// --- Comprobar que hay algo para generar
      L     "DB830_Dispositivos".Dispositivos[#NumeroDispositivo].StatusActual;
      L     0;
      ==I;
      JC    Final_GeneradorDeEmisiones;

      L     "Evento_DISPOSITIVO_EstadoActual";  // 160 - Refresco de Estado del Dispositivo
      T     "DB830_Dispositivos".Dispositivos[#NumeroDispositivo].EstadoEmisionEvento;
      JU    Final_GeneradorDeEmisiones;



NETWORK
TITLE = ---- Tratar ---> Cambio de Estado del Dispositivo
Tratar_CambioEstadoDeDispositivo:NOP   0;

////////////////////////////////////////////////////////////////////////////////////////
////////////////////////////////////////////////////////////////////////////////////////
////////////////////////////////////////////////////////////////////////////////////////
// --- Activar Evento (160) - Refresco del Estado del Dispositivo
      L     "DB830_Dispositivos".Dispositivos[#NumeroDispositivo].StatusReal;
      T     "DB830_Dispositivos".Dispositivos[#NumeroDispositivo].StatusActual;
      L     "DB830_Dispositivos".Dispositivos[#NumeroDispositivo].ErrorReal;
      T     "DB830_Dispositivos".Dispositivos[#NumeroDispositivo].ErrorActual;

      L     "Evento_DISPOSITIVO_EstadoActual";  // 160 - Refresco de Estado del Dispositivo
      T     "DB830_Dispositivos".Dispositivos[#NumeroDispositivo].EstadoEmisionEvento;

      JU    Final_GeneradorDeEmisiones;



NETWORK
TITLE = Generacion de Eventos
GeneradorDeEventos:NOP   0;

////////////////////////////////////////////////////////////////////////////////////////
////////////////////////////////////////////////////////////////////////////////////////
////////////////////////////////////////////////////////////////////////////////////////
// --- Existen Eventos a Emitir
      L     "DB830_Dispositivos".Dispositivos[#NumeroDispositivo].EstadoEmisionEvento;
      L     0;
      ==I;
      JC    Final_GeneradorDeEventos;


////////////////////////////////////////////////////////////////////////////////////////
////////////////////////////////////////////////////////////////////////////////////////
////////////////////////////////////////////////////////////////////////////////////////
// --- Variables para la Emision de Eventos (Depende del JDT)
      L     "JDT1_NDB_EventosEmi";
      T     #DBEventos;
      T     #NumDBEventos;
      L     "JDT1_MaxBytes";
      T     #MaxBytesDeEventos;

      SET;
      AN    "DB855_DefinicionDispositivos".Dispositivos[#NumeroDispositivo].EventosDelJdT02;
      JN    NoEsDispositivo_JDT02;

      L     "JDT2_NDB_EventosEmi";
      T     #DBEventos;
      T     #NumDBEventos;
      L     "JDT2_MaxBytes";
      T     #MaxBytesDeEventos;

NoEsDispositivo_JDT02:NOP   0;


////////////////////////////////////////////////////////////////////////////////////////
////////////////////////////////////////////////////////////////////////////////////////
////////////////////////////////////////////////////////////////////////////////////////
// --- Hay espacio para la Emision de Eventos
      L     0;
      T     #NumBytes;  // Inicializo el numero de Bytes
      LAR2;  // Inicializo el puntero de Eventos Generados

////////////////////////////////////////////////////////////////////////////////////////
// --- Calcula el tamaño de bytes que hay en el DB Eventos Generados

      OPN   DB [#DBEventos];
InicioBucleBusquedaFin_BufferEventos:NOP   0;
      L     DBB [AR2, P#0.0];
      L     0;
      ==I;  // Buscamos el final del DB = 0
      JC    FinalBucleBusquedaFin_BufferEventos;

      +AR2  P#1.0;
      JU    InicioBucleBusquedaFin_BufferEventos;

FinalBucleBusquedaFin_BufferEventos:NOP   0;
      TAR2;  // Guardo el puntero
      T     #P_Eventos;  // Sacamos el NumBytes Escritos
      SRD   3;
      T     #NumBytes;

////////////////////////////////////////////////////////////////////////////////////////
// --- Comprobamos si hay sitio para mas Eventos

      L     #NumBytes;  // Miramos si hay sitio
      L     #MaxBytesDeEventos;  // Max. que se pueden emitir, parametro
      >I;  // No se pueden generar más eventos
      JC    Final_GeneradorDeEventos;


////////////////////////////////////////////////////////////////////////////////////////
////////////////////////////////////////////////////////////////////////////////////////
////////////////////////////////////////////////////////////////////////////////////////
// --- Distribuir Segun Evento a Emitir


////////////////////////////////////////////////////////////////////////////////////////
// --- Estado del Dispositivo
      L     "DB830_Dispositivos".Dispositivos[#NumeroDispositivo].EstadoEmisionEvento;
      L     "Evento_DISPOSITIVO_EstadoActual";
      ==I;
      JC    GenerarEvento_EstadoDispositivo;


////////////////////////////////////////////////////////////////////////////////////////
// --- Fin de Reset
      L     "DB830_Dispositivos".Dispositivos[#NumeroDispositivo].EstadoEmisionEvento;
      L     "Evento_DISPOSITIVO_FinReset_OK";
      ==I;
      JC    GenerarEvento_FinResetProcesoDispositivo;
      L     "DB830_Dispositivos".Dispositivos[#NumeroDispositivo].EstadoEmisionEvento;
      L     "Evento_DISPOSITIVO_FinReset_NOK";
      ==I;
      JC    GenerarEvento_FinResetProcesoDispositivo;


////////////////////////////////////////////////////////////////////////////////////////
// --- Fin de Paro Blando
      L     "DB830_Dispositivos".Dispositivos[#NumeroDispositivo].EstadoEmisionEvento;
      L     "Evento_DISPOSITIVO_FinParoBlando_OK";
      ==I;
      JC    GenerarEvento_FinParoBlandoProcesoDispositivo;
      L     "DB830_Dispositivos".Dispositivos[#NumeroDispositivo].EstadoEmisionEvento;
      L     "Evento_DISPOSITIVO_FinParoBlando_NOK";
      ==I;
      JC    GenerarEvento_FinParoBlandoProcesoDispositivo;


////////////////////////////////////////////////////////////////////////////////////////
////////////////////////////////////////////////////////////////////////////////////////
////////////////////////////////////////////////////////////////////////////////////////
// --- Evento a Emitir NO VALIDO
      L     0;
      T     "DB830_Dispositivos".Dispositivos[#NumeroDispositivo].EstadoEmisionEvento;
      JU    Final_GeneradorDeEventos;


////////////////////////////////////////////////////////////////////////////////////////
////////////////////////////////////////////////////////////////////////////////////////
////////////////////////////////////////////////////////////////////////////////////////
// --- Fase Final - No hay que hacer mas en la Generacion de Eventos
Final_GeneradorDeEventos:NOP   0;
      BE;  // Finalizar Funcion



NETWORK
TITLE = ---- Generar el Evento STAT --> Estado del Dispositivo
GenerarEvento_EstadoDispositivo:NOP   0;

////////////////////////////////////////////////////////////////////////////////////////
////////////////////////////////////////////////////////////////////////////////////////
////////////////////////////////////////////////////////////////////////////////////////
// --- Evento de Dispositivo - Estado de Dispositivo - STAT
      LAR2  #P_Eventos;  // Puntero al DB de Eventos Generados

// --- Separacion entre Eventos a Generar
      L     #P_Eventos;  // Mirar si es el primer evento de la lista
      L     0;  // Es el primero ?
      ==I;
      JC    InicioBuffer_EventoSTAT_EstadoDispositivo;

      OPN   DB [#DBEventos];
      L     ',';  // Separador entre eventos ','
      T     DBB [AR2, P#0.0];
      +AR2  P#1.0;

InicioBuffer_EventoSTAT_EstadoDispositivo:NOP   0;


////////////////////////////////////////////////////////////////////////////////////////
////////////////////////////////////////////////////////////////////////////////////////
////////////////////////////////////////////////////////////////////////////////////////
// --- Inicio de Evento
      OPN   DB [#DBEventos];  // DB de Eventos Generados (A Emitir)
      L     '{';  // Inicio de Evento '{'
      T     DBB [AR2, P#0.0];
      +AR2  P#1.0;

      L     'STAT';  // Evento 'STAT'
      T     DBD [AR2, P#0.0];
      +AR2  P#4.0;


////////////////////////////////////////////////////////////////////////////////////////
// --- Atributo Tipo '[TIPO]'

      OPN   DB [#DBEventos];
      L     '[';
      T     DBB [AR2, P#0.0];
      L     'TIPO';
      T     DBD [AR2, P#1.0];
      L     ']';
      T     DBB [AR2, P#5.0];
      +AR2  P#6.0;

      L     'CBOX';
      T     DBD [AR2, P#0.0];
      +AR2  P#4.0;

////////////////////////////////////////////////////////////////////////////////////////
// --- Atributo Numero de Dispositivo '[NUME]'
      OPN   DB [#DBEventos];
      L     '[';
      T     DBB [AR2, P#0.0];
      L     'NUME';
      T     DBD [AR2, P#1.0];
      L     ']';
      T     DBB [AR2, P#5.0];
      +AR2  P#6.0;

      L     "CTE_OffsetCCPIF";
      L     1;
      +I;
      L     100;
      *I;
      L     #NumeroDispositivo;  // Numero de Dispo
      +I;
      T     #Valor;

// --- Convertir Valor a ASCII - Numero de Dispositivo
      TAR2;
      SRD   3;
      T     #OffsetInicial;  // Miro que offset tiene la String

      CALL  "FC893_Obtener_StringDelAtributo"
      ( DB_String := #NumDBEventos,
        OffsetIni := #OffsetInicial,
        Valor     := #Valor,
        OffsetFin := #OffsetFinal
      );  // Llamo a ObtenerStrinAtributo

      L     #OffsetFinal;
      SLD   3;
      LAR2;  // Recupero que offset tiene la String


////////////////////////////////////////////////////////////////////////////////////////
// --- Atributo Numero de Dispositivo '[NUES]'
      OPN   DB [#DBEventos];
      L     '[';
      T     DBB [AR2, P#0.0];
      L     'NUES';
      T     DBD [AR2, P#1.0];
      L     ']';
      T     DBB [AR2, P#5.0];
      +AR2  P#6.0;

      L     "DB830_Dispositivos".Dispositivos[#NumeroDispositivo].StatusActual;
      L     W#16#F;  // Solo la parte Estado
      AW;
      T     #Convertir;

      CALL  "FC895_Obtener_EtiquetaDeValor"
      ( ValorEvento    := #Convertir,
        EtiquetaEvento := #Conversion
      );

      OPN   DB [#DBEventos];
      L     #Conversion;
      T     DBD [AR2, P#0.0];
      +AR2  P#4.0;


////////////////////////////////////////////////////////////////////////////////////////
// --- Atributo Numero de Dispositivo '[LLAV]'
      OPN   DB [#DBEventos];
      L     '[';  // Evento -
      T     DBB [AR2, P#0.0];
      L     'LLAV';
      T     DBD [AR2, P#1.0];
      L     ']';
      T     DBB [AR2, P#5.0];
      +AR2  P#6.0;

      L     "DB830_Dispositivos".Dispositivos[#NumeroDispositivo].StatusActual;
      L     W#16#F0;  // Solo la parte Llave
      AW;
      SRD   4;
      L     10;
      +I;
      T     #Convertir;

      T     #Convertir;
      CALL  "FC895_Obtener_EtiquetaDeValor"
      ( ValorEvento    := #Convertir,
        EtiquetaEvento := #Conversion
      );

      OPN   DB [#DBEventos];
      L     #Conversion;
      T     DBD [AR2, P#0.0];
      +AR2  P#4.0;


////////////////////////////////////////////////////////////////////////////////////////
// --- Poner Error (Si es necesario)
      L     "DB830_Dispositivos".Dispositivos[#NumeroDispositivo].ErrorActual;
      L     0;
      ==D;
      JC    NoErrorDispositivo_STAT_EstadoDispositivo;


// --- Atributo Numero de Dispositivo '[CODE]'
      OPN   DB [#DBEventos];
      L     '[';  // Evento -
      T     DBB [AR2, P#0.0];
      L     'CODE';
      T     DBD [AR2, P#1.0];
      L     ']';
      T     DBB [AR2, P#5.0];
      +AR2  P#6.0;

      L     "DB830_Dispositivos".Dispositivos[#NumeroDispositivo].ErrorActual;
      T     #Valor;

// --- Convertir Valor a ASCII - Error
      TAR2;
      SRD   3;
      T     #OffsetInicial;  // Miro que offset tiene la String

      CALL  "FC893_Obtener_StringDelAtributo"
      ( DB_String := #NumDBEventos,
        OffsetIni := #OffsetInicial,
        Valor     := #Valor,
        OffsetFin := #OffsetFinal
      );  // Llamo a ObtenerStrinAtributo

      L     #OffsetFinal;
      SLD   3;
      LAR2;  // Recupero que offset tiene la String

NoErrorDispositivo_STAT_EstadoDispositivo:NOP   0;


////////////////////////////////////////////////////////////////////////////////////////
// --- Final del formaateo del Evento
      OPN   DB [#DBEventos];  // DB de Eventos Generados (A Emitir)
      L     '}';  // Fin de Evento '}'
      T     DBB [AR2, P#0.0];
      +AR2  P#1.0;


////////////////////////////////////////////////////////////////////////////////////////
////////////////////////////////////////////////////////////////////////////////////////
////////////////////////////////////////////////////////////////////////////////////////
// --- Dar por formateado el Evento

      L     0;  // 0 - Lo doy por tratado
      T     "DB830_Dispositivos".Dispositivos[#NumeroDispositivo].EstadoEmisionEvento;

      JU    Final_GeneradorDeEventos;



NETWORK
TITLE = ---- Generar el Evento FIN! --> Reset OK, Reset NOK
GenerarEvento_FinResetProcesoDispositivo:NOP   0;

////////////////////////////////////////////////////////////////////////////////////////
////////////////////////////////////////////////////////////////////////////////////////
////////////////////////////////////////////////////////////////////////////////////////
// --- Formateo del Evento FIN! (Fin del Proceso --> Reset y Paro Blando)
      LAR2  #P_Eventos;  // Puntero al DB de Eventos Generados

// --- Separacion entre Eventos a Generar
      L     #P_Eventos;  // Mirar si es el primer evento de la lista
      L     0;  // Es el primero ?
      ==I;
      JC    InicioBuffer_EventoFIN_FinResetProcesoDispositivo;

      OPN   DB [#DBEventos];
      L     ',';  // Separador entre eventos ','
      T     DBB [AR2, P#0.0];
      +AR2  P#1.0;

InicioBuffer_EventoFIN_FinResetProcesoDispositivo:NOP   0;


////////////////////////////////////////////////////////////////////////////////////////
////////////////////////////////////////////////////////////////////////////////////////
////////////////////////////////////////////////////////////////////////////////////////
// --- Inicio de Evento
      OPN   DB [#DBEventos];  // DB de Eventos Generados (A Emitir)
      L     '{';  // Inicio de Evento '{'
      T     DBB [AR2, P#0.0];
      +AR2  P#1.0;

      L     'FIN!';  // Evento 'FIN!'
      T     DBD [AR2, P#0.0];
      +AR2  P#4.0;


////////////////////////////////////////////////////////////////////////////////////////
// --- Atributo Tipo '[TIPO]'

      OPN   DB [#DBEventos];
      L     '[';
      T     DBB [AR2, P#0.0];
      L     'TIPO';
      T     DBD [AR2, P#1.0];
      L     ']';
      T     DBB [AR2, P#5.0];
      +AR2  P#6.0;


      L     'CBOX';
      T     DBD [AR2, P#0.0];
      +AR2  P#4.0;

////////////////////////////////////////////////////////////////////////////////////////
// --- Atributo Numero de Dispositivo '[NUME]'
      OPN   DB [#DBEventos];
      L     '[';
      T     DBB [AR2, P#0.0];
      L     'NUME';
      T     DBD [AR2, P#1.0];
      L     ']';
      T     DBB [AR2, P#5.0];
      +AR2  P#6.0;

      L     "CTE_OffsetCCPIF";
      L     1;
      +I;
      L     100;
      *I;
      L     #NumeroDispositivo;  // Numero de Dispo
      +I;
      T     #Valor;

// --- Convertir Valor a ASCII - Numero de Dispositivo
      TAR2;
      SRD   3;
      T     #OffsetInicial;  // Miro que offset tiene la String

      CALL  "FC893_Obtener_StringDelAtributo"
      ( DB_String := #NumDBEventos,
        OffsetIni := #OffsetInicial,
        Valor     := #Valor,
        OffsetFin := #OffsetFinal
      );  // Llamo a ObtenerStrinAtributo

      L     #OffsetFinal;
      SLD   3;
      LAR2;  // Recupero que offset tiene la String


////////////////////////////////////////////////////////////////////////////////////////
// --- Atributo Numero de Dispositivo '[PROC]'
      OPN   DB [#DBEventos];
      L     '[';
      T     DBB [AR2, P#0.0];
      L     'PROC';
      T     DBD [AR2, P#1.0];
      L     ']';
      T     DBB [AR2, P#5.0];
      +AR2  P#6.0;

      OPN   DB [#DBEventos];
      L     'RESE';
      T     DBD [AR2, P#0.0];
      +AR2  P#4.0;


////////////////////////////////////////////////////////////////////////////////////////
// --- Atributo Numero de Dispositivo '[RSLT]'
      OPN   DB [#DBEventos];
      L     '[';
      T     DBB [AR2, P#0.0];
      L     'RSLT';
      T     DBD [AR2, P#1.0];
      L     ']';
      T     DBB [AR2, P#5.0];
      +AR2  P#6.0;

      L     "DB830_Dispositivos".Dispositivos[#NumeroDispositivo].EstadoEmisionEvento;
      L     151;
      -I;
      L     W#16#30;  // Convertir a ASCII
      +I;
      OPN   DB [#DBEventos];
      T     DBB [AR2, P#0.0];
      +AR2  P#1.0;


////////////////////////////////////////////////////////////////////////////////////////
// --- Final del formaateo del Evento
      OPN   DB [#DBEventos];  // DB de Eventos Generados (A Emitir)
      L     '}';  // Fin de Evento '}'
      T     DBB [AR2, P#0.0];
      +AR2  P#1.0;


////////////////////////////////////////////////////////////////////////////////////////
////////////////////////////////////////////////////////////////////////////////////////
////////////////////////////////////////////////////////////////////////////////////////
// --- Dar por formateado el Evento

      L     0;  // 0 - Lo doy por tratado
      T     "DB830_Dispositivos".Dispositivos[#NumeroDispositivo].EstadoEmisionEvento;

      JU    Final_GeneradorDeEventos;




NETWORK
TITLE = ---- Generar el Evento FIN! --> ParoBlando OK ParoBlandoNOK
GenerarEvento_FinParoBlandoProcesoDispositivo:NOP   0;

////////////////////////////////////////////////////////////////////////////////////////
////////////////////////////////////////////////////////////////////////////////////////
////////////////////////////////////////////////////////////////////////////////////////
// --- Formateo del Evento FIN! (Fin del Proceso --> Reset y Paro Blando)
      LAR2  #P_Eventos;  // Puntero al DB de Eventos Generados

// --- Separacion entre Eventos a Generar
      L     #P_Eventos;  // Mirar si es el primer evento de la lista
      L     0;  // Es el primero ?
      ==I;
      JC    InicioBuffer_EventoFIN_FinParoBlandoProcesoDispositivo;

      OPN   DB [#DBEventos];
      L     ',';  // Separador entre eventos ','
      T     DBB [AR2, P#0.0];
      +AR2  P#1.0;

InicioBuffer_EventoFIN_FinParoBlandoProcesoDispositivo:NOP   0;


////////////////////////////////////////////////////////////////////////////////////////
////////////////////////////////////////////////////////////////////////////////////////
////////////////////////////////////////////////////////////////////////////////////////
// --- Inicio de Evento
      OPN   DB [#DBEventos];  // DB de Eventos Generados (A Emitir)
      L     '{';  // Inicio de Evento '{'
      T     DBB [AR2, P#0.0];
      +AR2  P#1.0;

      L     'FIN!';  // Evento 'FIN!'
      T     DBD [AR2, P#0.0];
      +AR2  P#4.0;


////////////////////////////////////////////////////////////////////////////////////////
// --- Atributo Tipo '[TIPO]'

      OPN   DB [#DBEventos];
      L     '[';
      T     DBB [AR2, P#0.0];
      L     'TIPO';
      T     DBD [AR2, P#1.0];
      L     ']';
      T     DBB [AR2, P#5.0];
      +AR2  P#6.0;


      L     'CBOX';
      T     DBD [AR2, P#0.0];
      +AR2  P#4.0;

////////////////////////////////////////////////////////////////////////////////////////
// --- Atributo Numero de Dispositivo '[NUME]'
      OPN   DB [#DBEventos];
      L     '[';
      T     DBB [AR2, P#0.0];
      L     'NUME';
      T     DBD [AR2, P#1.0];
      L     ']';
      T     DBB [AR2, P#5.0];
      +AR2  P#6.0;

      L     "CTE_OffsetCCPIF";
      L     1;
      +I;
      L     100;
      *I;
      L     #NumeroDispositivo;  // Numero de Dispo
      +I;
      T     #Valor;

// --- Convertir Valor a ASCII - Numero de Dispositivo
      TAR2;
      SRD   3;
      T     #OffsetInicial;  // Miro que offset tiene la String

      CALL  "FC893_Obtener_StringDelAtributo"
      ( DB_String := #NumDBEventos,
        OffsetIni := #OffsetInicial,
        Valor     := #Valor,
        OffsetFin := #OffsetFinal
      );  // Llamo a ObtenerStrinAtributo

      L     #OffsetFinal;
      SLD   3;
      LAR2;  // Recupero que offset tiene la String


////////////////////////////////////////////////////////////////////////////////////////
// --- Atributo Numero de Dispositivo '[PROC]'
      OPN   DB [#DBEventos];
      L     '[';
      T     DBB [AR2, P#0.0];
      L     'PROC';
      T     DBD [AR2, P#1.0];
      L     ']';
      T     DBB [AR2, P#5.0];
      +AR2  P#6.0;

      OPN   DB [#DBEventos];
      L     'BLAN';
      T     DBD [AR2, P#0.0];
      +AR2  P#4.0;


////////////////////////////////////////////////////////////////////////////////////////
// --- Atributo Numero de Dispositivo '[RSLT]'
      OPN   DB [#DBEventos];
      L     '[';
      T     DBB [AR2, P#0.0];
      L     'RSLT';
      T     DBD [AR2, P#1.0];
      L     ']';
      T     DBB [AR2, P#5.0];
      +AR2  P#6.0;

      L     "DB830_Dispositivos".Dispositivos[#NumeroDispositivo].EstadoEmisionEvento;
      L     153;
      -I;
      L     W#16#30;  // Convertir a ASCII
      +I;
      OPN   DB [#DBEventos];
      T     DBB [AR2, P#0.0];
      +AR2  P#1.0;


////////////////////////////////////////////////////////////////////////////////////////
// --- Final del formaateo del Evento
      OPN   DB [#DBEventos];  // DB de Eventos Generados (A Emitir)
      L     '}';  // Fin de Evento '}'
      T     DBB [AR2, P#0.0];
      +AR2  P#1.0;


////////////////////////////////////////////////////////////////////////////////////////
////////////////////////////////////////////////////////////////////////////////////////
////////////////////////////////////////////////////////////////////////////////////////
// --- Dar por formateado el Evento

      L     0;  // 0 - Lo doy por tratado
      T     "DB830_Dispositivos".Dispositivos[#NumeroDispositivo].EstadoEmisionEvento;

      JU    Final_GeneradorDeEventos;



END_FUNCTION

FUNCTION "FC755_EventosApilaDesApila" : Void   // FC755, STL
TITLE = Emision de los Eventos del Apilador-DesApialdor
{ S7_Optimized_Access := 'FALSE' }
AUTHOR : TRACKING
NAME : 20141014
VERSION : 4.0
// stored: AutoNumber false
   VAR_INPUT
      NumMaquina : UInt;   // Numero de Maquina
      EstadoMaquina : "EstadoZona";   // Estado de la Maquina
      EstadoVIMaquina : "EstadoMaquina";   // Estado del VI de la Maquina
      ApiladorVacio : Bool;   // Apilador esta Vacio
      ApiladorSemiLleno : Bool;   // Apilador esta SemiLleno
      ApiladorLleno : Bool;   // Apilador esta LLeno
      MesaDeJDT02 : Bool;
   END_VAR
   VAR_TEMP
      EstadoActual : UInt;
      P_EmiEventos : DWord;
      DBEventos : Word;
      NumBytes : UInt;
      OffsetInicial : UInt;
      OffsetFinal : UInt;
      Conversion : DWord;
      Convertir : UInt;
      Valor : UDInt;
      NumDBEventos : UInt;
      MaxBytes : UInt;
   END_VAR
BEGIN

NETWORK
TITLE = Inicializaciones
///////////////////////////////////////////////////////////////////////////////
/// Inicio --> Pertenece al JDT 02

      L     "JDT1_NDB_EventosEmi";
      T     #DBEventos;
      T     #NumDBEventos;
      L     "JDT1_MaxBytes";
      T     #MaxBytes;

      AN    #MesaDeJDT02;
      JC    NoJdT02;

      L     "JDT2_NDB_EventosEmi";
      T     #DBEventos;
      T     #NumDBEventos;
      L     "JDT2_MaxBytes";
      T     #MaxBytes;

NoJdT02:NOP   0;

/// Final --> Pertenece al JDT 02
///////////////////////////////////////////////////////////////////////////////




NETWORK
TITLE = Mirar si se pueden generar eventos
// - Inicializo el Numero de Bytes y el puntero del DB de Eventos Generados
// - Calcula el Tamaño de bytes que hay en el DB de Eventos Genardos
// - Comprobamos si hay sitio para Eventos
///////////////////////////////////////////////////////////////////////////////
/// Inicializo el Numero de Bytes y el puntero del DB Eventos Generados

      L     0;
      T     #NumBytes;  // Inicializo el numero de Bytes
      LAR2;  // Inicializo el puntero de Eventos Generados

///////////////////////////////////////////////////////////////////////////////
/// Calcula el tamaño de bytes que hay en el DB Eventos Generados

      OPN   DB [#DBEventos];

Inicio_BusquedaFinalEventos:NOP   0;
      L     DBB [AR2, P#0.0];
      L     0;
      ==I;
      JC    Final_BusquedaFinalEventos;  // Buscamos el final del DB = 0

      +AR2  P#1.0;
      JU    Inicio_BusquedaFinalEventos;

Final_BusquedaFinalEventos:NOP   0;
      TAR2;  // Guardo el puntero
      T     #P_EmiEventos;  // Sacamos el NumBytes Escritos
      SRD   3;
      T     #NumBytes;

// -----------------------------------------------------------------------------------------------
// Comprobamos si hay sitio para mas Eventos

      L     #NumBytes;  // Miramos si hay sitio
      L     #MaxBytes;  // Max. que se pueden emitir, parametro
      >I;
      JC    Final;  // No se pueden generar más eventos


NETWORK
TITLE = Distribucion
///////////////////////////////////////////////////////////////////////////////
// --- Distribucion  del Estado de Trabajo del Apilador

      L     0;
      T     #EstadoActual;

// ---------- Mirar si esta Vacio el Apilador

      A     #ApiladorVacio;
      AN    #ApiladorSemiLleno;
      AN    #ApiladorLleno;
      JCN   _ST1;  // No Esta Vacio ?

      L     1000;  // Esta Vacio
      T     #EstadoActual;
      JU    _STF;


// ---------- Mirar si esta Semi-Lleno el Apilador

_ST1: AN    #ApiladorVacio;
      A     #ApiladorSemiLleno;
      AN    #ApiladorLleno;
      JCN   _ST2;  // No Esta Semi-Lleno ?

      L     1001;  // Esta Semi-Lleno
      T     #EstadoActual;
      JU    _STF;


// ---------- Mirar si esta Lleno el Apilador

_ST2: AN    #ApiladorVacio;
      AN    #ApiladorSemiLleno;
      A     #ApiladorLleno;
      JCN   _ST3;  // No Esta Lleno ?

      L     1002;  // Esta Lleno
      T     #EstadoActual;
      JU    _STF;


// ---------- No se sabe como esta el apilador

_ST3: L     0;  // No se Sabe el Status de Trabajo
      T     "DB832_Maquinas".Maquinas[#NumMaquina].MemoriaEstado;

      JU    ST_F;


///////////////////////////////////////////////////////////////////////////////
// ---------- Mirar si hay que Emitir el Evento

_STF: L     "DB832_Maquinas".Maquinas[#NumMaquina].Operacion;
      L     5000;  // Peticion de Status del Apilador
      <>I;
      JC    ST_F;

      L     #EstadoActual;
      L     0;  // Existe Status del Apilador
      ==I;
      JC    ST_F;

      JU    EmisionDelEvento;


///////////////////////////////////////////////////////////////////////////////
// --- Fin del Estado de Trabajo del Apilador

ST_F: JU    Final;



NETWORK
TITLE = Emision del Evento
///////////////////////////////////////////////////////////////////////////////
// --- Formateo del Evento DIDA - Estado del Apilador - DesApilador

EmisionDelEvento:NOP   0;
      L     #P_EmiEventos;
      LAR2;  // Puntero al DB de Eventos Generados

      TAR2;  // Mirar si es el primer evento de la lista
      L     0;
      ==I;
      JC    NoEsInicio_ListaDeEventos;  // Es el primero

      OPN   DB [#DBEventos];
      L     ',';  // Separador entre eventos ','
      T     DBB [AR2, P#0.0];
      +AR2  P#1.0;

NoEsInicio_ListaDeEventos:NOP   0;
      OPN   DB [#DBEventos];  // DB de Eventos Generados (A Emitir)
      L     '{';  // Inicio de Evento '{'
      T     DBB [AR2, P#0.0];
      +AR2  P#1.0;


///////////////////////////////////////////////////////////////////////////////
// --- Cuerpo del Evento

      L     'DIDA';  // Evento 'DIDA'
      T     DBD [AR2, P#0.0];
      +AR2  P#4.0;

      OPN   DB [#DBEventos];
      L     '[';  // Evento - Atributo Tipo '[TIPO]'
      T     DBB [AR2, P#0.0];
      L     'TIPO';
      T     DBD [AR2, P#1.0];
      L     ']';
      T     DBB [AR2, P#5.0];
      +AR2  P#6.0;

      L     "DB850_DefinicionMesas".Mesa[#NumMaquina].ConfigMesa.TipoMaquina;
      T     #Convertir;

      CALL  "FC895_Obtener_EtiquetaDeValor"
      ( ValorEvento    := #Convertir,
        EtiquetaEvento := #Conversion
      );

      OPN   DB [#DBEventos];
      L     #Conversion;
      T     DBD [AR2, P#0.0];
      +AR2  P#4.0;


      L     '[';  // Evento - Atributo Numero de Dispositivo '[NUME]'
      T     DBB [AR2, P#0.0];
      L     'NUME';
      T     DBD [AR2, P#1.0];
      L     ']';
      T     DBB [AR2, P#5.0];
      +AR2  P#6.0;

      L     "CTE_OffsetMesa";
      L     #NumMaquina;  // Numero de Maquina
      +I;
      T     #Valor;

// --- Convertir Valor a ASCII - Numero de Maquina
      TAR2;
      SRD   3;
      T     #OffsetInicial;  // Miro que offset tiene la String

      CALL  "FC893_Obtener_StringDelAtributo"
      ( DB_String := #NumDBEventos,
        OffsetIni := #OffsetInicial,
        Valor     := #Valor,
        OffsetFin := #OffsetFinal
      );  // Llamo a ObtenerStrinAtributo

      L     #OffsetFinal;
      SLD   3;
      LAR2;  // Recupero que offset tiene la String

// --- Ya esta convertido el Valor a ASCII

      OPN   DB [#DBEventos];
      L     '[';  // Evento - Atributo Numero de Dispositivo '[FULL]'
      T     DBB [AR2, P#0.0];
      L     'FULL';
      T     DBD [AR2, P#1.0];
      L     ']';
      T     DBB [AR2, P#5.0];
      +AR2  P#6.0;

      L     #EstadoActual;  // Estado Actual del Apilador
      T     #Convertir;

      CALL  "FC895_Obtener_EtiquetaDeValor"
      ( ValorEvento    := #Convertir,
        EtiquetaEvento := #Conversion
      );

      OPN   DB [#DBEventos];
      L     #Conversion;
      T     DBD [AR2, P#0.0];
      +AR2  P#4.0;


///////////////////////////////////////////////////////////////////////////////
// Final del formateo del Evento

      OPN   DB [#DBEventos];  // DB de Eventos Generados (A Emitir)
      L     '}';  // Fin de Evento '}'
      T     DBB [AR2, P#0.0];
      +AR2  P#1.0;

///////////////////////////////////////////////////////////////////////////////
// Dar por formateado el Evento

      L     #EstadoActual;  // Lo doy por tratado
      T     "DB832_Maquinas".Maquinas[#NumMaquina].MemoriaEstado;
      L     0;
      T     "DB832_Maquinas".Maquinas[#NumMaquina].Operacion;

      JU    Final;  // Ya se ha generado el evento de la Maquina

// Fin del Formateo del Evento DIDA (Apilador)
///////////////////////////////////////////////////////////////////////////////
///////////////////////////////////////////////////////////////////////////////



NETWORK
TITLE = Fin de la Funcion
///////////////////////////////////////////////////////////////////////////////
//// -- Final de la Funcion
Final:NOP   0;



END_FUNCTION

FUNCTION "FC776_Presion_DesPaletizador_Paletizador_Automatico" : Void   // FC776, STL
TITLE = Calculo de Presion del DesPaletizador
{ S7_Optimized_Access := 'FALSE' }
AUTHOR : TRACKING
NAME : 20130301
VERSION : 3.0
// stored: AutoNumber false
   VAR_INPUT
      Mesa : UInt;   // Mesa del DesPaletizador
      CalcularPresion : Bool;   // Orden de Calcular la Presion
   END_VAR
   VAR_IN_OUT
      PresionUT : Word;   // Presion ha utilizar para la UT de la Mesa
      FinCalculoPresion : Bool;   // Ya Realizado el Calculo de la Presion
   END_VAR
   VAR_TEMP
      NumeroUT : UInt;
   END_VAR
BEGIN

NETWORK
TITLE = Distribucion
////////////////////////////////////////////////////////////////////////////
// --- DISTRIBUCION
// ---

      AN    #FinCalculoPresion;
      A     #CalcularPresion;
      JC    CalcularDePresion;  // Calcular la Presion ?

      A     #FinCalculoPresion;
      AN    #CalcularPresion;
      JC    Fin_CalculoDePresion;  // Cierre de Protocolo ?

      BE;  // - Finalizar del Bloque



NETWORK
TITLE = Calcular la Presion
////////////////////////////////////////////////////////////////////////////
// --- CALCULAR LA PRESION
// ---
// --- Buscar la primera UT de la Mesa
// --- Recoger la Presion de la UT de la Base de Datos
// --- Dar por finalizado el Caculo, Activando el Protocolo
// ---

CalcularDePresion:NOP   0;
      L     "DB810_ColasMesas".Colas[#Mesa].UT_PrimeraMesa;
      T     #NumeroUT;

      SET;
      S     #FinCalculoPresion;  // Activar el Protocolo

// Presion para DesPaletizar y Paletizar
      L     "DB815_UTs_Datos".UT[#NumeroUT].Presion;
      T     #PresionUT;

      BE;  // - Finalizar del Bloque


////////////////////////////////////////////////////////////////////////////
// --- CIERRE DE PROTOCOLO
// ---

Fin_CalculoDePresion:NOP   0;

      SET;
      R     #FinCalculoPresion;  // - Cerrado el Protocolo
      L     0;
      T     #PresionUT;

      BE;  // - Finalizar del Bloque


END_FUNCTION

FUNCTION "FC791_GestorLlave" : Void   // FC791, LAD
{ S7_Optimized_Access := 'FALSE' }
AUTHOR : TRACKING
NAME : 20160411
VERSION : 3.1
// stored: AutoNumber false, SetENOAutomatically false
   VAR_INPUT
      NumLlave : UInt;
      Estado : Bool;
      MesaDeJDT02 : Bool;
   END_VAR
   VAR_OUTPUT
      Llave : "UDT_DatosLlave";
   END_VAR
   VAR_TEMP
      PunteroEventos : DWord;
      DBEventos : Word;
      NumDBEventos : UInt;
      MaxBytesDeEventos : UInt;
      NumBytes : UInt;
      Offset : UInt;   // Offset donde esta el Primer Dispositivo
      ValorTMP : UDInt;
      ValorReturn : Int;
   END_VAR
BEGIN

NETWORK
TITLE = Inicializar
////////////////////////////////////////////////////////////////////////////
// --- Inicializar Variables


////////////////////////////////////////////////////////////////////////////
// --- Control Numero de Dispositivo

      L     #NumLlave;
      L     1;
      <I;
      JC    FinalFuncion;  // Ha superado el minimo
      L     #NumLlave;
      L     "CTE_MaxDispositivosLlave";
      >I;
      JC    FinalFuncion;  // Ha superado el maximo



NETWORK
TITLE = Acciones
////////////////////////////////////////////////////////////////////////////
// --- Cambio de estado de la llave ?

      SET;
      A     #Estado;
      AN    "DB839_DispositivosVarios".DispoLlave[#NumLlave].EstadoActual;
      JC    CambioDeEstado_Llave;

      SET;
      AN    #Estado;
      A     "DB839_DispositivosVarios".DispoLlave[#NumLlave].EstadoActual;
      JC    CambioDeEstado_Llave;


////////////////////////////////////////////////////////////////////////////
// --- Mirar si hay peticion de Estado de Llave

      SET;
      A     "DB839_DispositivosVarios".DispoLlave[#NumLlave].RefrescoDatos;
      JC    EnviarEvento_RefrescoDeDatos;  // Hay Peticion de Esatdo ?
      JU    FinalFuncion;  // No Hay Peticion de estado



////////////////////////////////////////////////////////////////////////////
// --- Ha cambiado de estado la Llave

CambioDeEstado_Llave:NOP   0;
      SET;
      A     #Estado;  // Guardar el estado de la Llave
      =     "DB839_DispositivosVarios".DispoLlave[#NumLlave].EstadoActual;

      SET;
      S     "DB839_DispositivosVarios".DispoLlave[#NumLlave].RefrescoDatos;  // Activar la Peticion de Estado de la Llave

      JU    EnviarEvento_RefrescoDeDatos;  // Mandar nuevo evento de Estado de Llave



NETWORK
TITLE = Evento de Estado de la Llave
EnviarEvento_RefrescoDeDatos:NOP   0;

////////////////////////////////////////////////////////////////////////////
// ---   Formateo del Evento de Estado del Dispositivo
// ---   * Mirar si hay sitio para generar el nuevo evento
// ---       * Inicializo NumBytes y Puntero al DB de Eventos Generados
// ---       * Calcula el tamaño de bytes que hay en el DB de Eventos Generados
// ---       * Comprobar si hay sitio para un evento más
// ---   * Formatear el evento de Estado de las Llaves
////////////////////////////////////////////////////////////////////////////



////////////////////////////////////////////////////////////////////////////
// --- Inicio --> Pertenece a JDT 02 (Por defecto Pertenece a JDT01)

      L     "JDT1_NDB_EventosEmi";
      T     #DBEventos;
      T     #NumDBEventos;
      L     "JDT1_MaxBytes";
      T     #MaxBytesDeEventos;

      SET;
      AN    #MesaDeJDT02;
      JC    NoPerteneceJDT02;

      L     "JDT2_NDB_EventosEmi";
      T     #DBEventos;
      T     #NumDBEventos;
      L     "JDT2_MaxBytes";
      T     #MaxBytesDeEventos;

NoPerteneceJDT02:NOP   0;
// --- Fin --> Pertenece a JDT 02
////////////////////////////////////////////////////////////////////////////



////////////////////////////////////////////////////////////////////////////
// --- Mirar si hay sitio para generar un evento más

      L     0;
      T     #NumBytes;  // Inicializo el numero de Bytes
      T     #PunteroEventos;  // Inicializo el puntero de Eventos Generados

Inicio_BusquedaFinalEventos:NOP   0;
      OPN   DB [#DBEventos];  // Calcula el tamaño de bytes que hay en el DB
      L     DBB [#PunteroEventos];
      L     0;
      ==I;
      JC    Fin_BusquedaFinalEventos;  // Buscamos el final del DB = 0

      OPN   DB [#DBEventos];
      L     DBB [#PunteroEventos];
      L     ' ';
      ==I;
      JC    Fin_BusquedaFinalEventos;  // Buscamos el final del DB = ' '

      L     #PunteroEventos;  // Incremento de P#1.0
      L     P#1.0;
      +D;
      T     #PunteroEventos;

      JU    Inicio_BusquedaFinalEventos;  // Continuar con el siguiente posicion

Fin_BusquedaFinalEventos:NOP   0;
      L     #PunteroEventos;  // Sacamos el NumBytes Escritos
      SRD   3;
      T     #NumBytes;

      L     #NumBytes;  // Miramos si hay sitio
      L     #MaxBytesDeEventos;  // Max. que se pueden emitir, parametro
      >I;
      JC    FinalFuncion;  // No se pueden generar más eventos


////////////////////////////////////////////////////////////////////////////
// --- Formatear el evento de Estado del Dispositivo

      L     #PunteroEventos;
      LAR2;  // Puntero al DB de Eventos Generados

      TAR2;  // Mirar si es el primer evento de la lista
      L     0;
      ==I;
      JC    NoEsInicio_ListaDeEventos;  // Es el primero

      OPN   DB [#DBEventos];
      L     ',';  // Separador entre eventos ','
      T     DBB [AR2, P#0.0];
      +AR2  P#1.0;

NoEsInicio_ListaDeEventos:NOP   0;
      OPN   DB [#DBEventos];  // DB de Eventos Generados (A Emitir)
      L     '{';  // Inicio de Evento '{'
      T     DBB [AR2, P#0.0];
      +AR2  P#1.0;


////////////////////////////////////////////////////////////////////////////
      L     'STAT';  // --- Evento 'STAT'
      T     DBD [AR2, P#0.0];
      +AR2  P#4.0;


////////////////////////////////////////////////////////////////////////////
      OPN   DB [#DBEventos];
      L     '[';
      T     DBB [AR2, P#0.0];
      L     'TIPO';
      T     DBD [AR2, P#1.0];
      L     ']';
      T     DBB [AR2, P#5.0];
      +AR2  P#6.0;

      OPN   DB [#DBEventos];
      L     'LLAV';  // Tipo Llave
      T     DBD [AR2, P#0.0];
      +AR2  P#4.0;


////////////////////////////////////////////////////////////////////////////
      L     '[';
      T     DBB [AR2, P#0.0];
      L     'NUME';
      T     DBD [AR2, P#1.0];
      L     ']';
      T     DBB [AR2, P#5.0];
      +AR2  P#6.0;

      L     "CTE_OffsetMesa";
      L     #NumLlave;  // Numero de la Llave
      +I;
      T     #ValorTMP;

// --- Convertir Valor a ASCII - Numero de la Baliza
      TAR2;
      SRD   3;
      T     #NumBytes;  // Miro que offset tiene la String

      CALL  "FC893_Obtener_StringDelAtributo"
      ( DB_String := #NumDBEventos,
        OffsetIni := #NumBytes,
        Valor     := #ValorTMP,
        OffsetFin := #Offset
      );  // Llamo a ObtenerStrinAtributo

      L     #Offset;
      SLD   3;
      LAR2;  // Recupero que offset tiene la String

// --- Ya esta convertido el Valor a ASCII

////////////////////////////////////////////////////////////////////////////
      OPN   DB [#DBEventos];
      L     '[';
      T     DBB [AR2, P#0.0];
      L     'ACTI';
      T     DBD [AR2, P#1.0];
      L     ']';
      T     DBB [AR2, P#5.0];
      +AR2  P#6.0;

      L     'SI';
      SET;
      A     "DB839_DispositivosVarios".DispoLlave[#NumLlave].EstadoActual;  // Activo Llave ?
      JC    EstaActiva_Llave;
      L     'NO';
EstaActiva_Llave:NOP   0;
      OPN   DB [#DBEventos];
      T     DBW [AR2, P#0.0];
      +AR2  P#2.0;


////////////////////////////////////////////////////////////////////////////
      OPN   DB [#DBEventos];
      L     '[';
      T     DBB [AR2, P#0.0];
      L     'HABI';
      T     DBD [AR2, P#1.0];
      L     ']';
      T     DBB [AR2, P#5.0];
      +AR2  P#6.0;

      L     'SI';
      SET;
      A     "DB839_DispositivosVarios".DispoLlave[#NumLlave].Habilitado;  // Habilitado ?
      JC    EstaDesHabilitada_Llave;
      L     'NO';
EstaDesHabilitada_Llave:NOP   0;
      OPN   DB [#DBEventos];
      T     DBW [AR2, P#0.0];
      +AR2  P#2.0;


////////////////////////////////////////////////////////////////////////////
      OPN   DB [#DBEventos];  // DB de Eventos Generados (A Emitir)
      L     '}';  // --- Fin de Evento '}'
      T     DBB [AR2, P#0.0];
      +AR2  P#1.0;



////////////////////////////////////////////////////////////////////////////
// --- Final del Evento

      SET;
      R     "DB839_DispositivosVarios".DispoLlave[#NumLlave].RefrescoDatos;  // Activar la Peticion de Estado de la Baliza

      JU    FinalFuncion;  //Final del Formateo del Elento



NETWORK
TITLE = Final de la Función
////////////////////////////////////////////////////////////////////////////
FinalFuncion:NOP   0;

      CALL  BLKMOV
      ( SRCBLK  := "DB839_DispositivosVarios".DispoLlave[#NumLlave],
        RET_VAL := #ValorReturn,
        DSTBLK  := #Llave
      );


END_FUNCTION

FUNCTION "FC792_GestorSeta" : Void   // FC792, LAD
{ S7_Optimized_Access := 'FALSE' }
AUTHOR : TRACKING
NAME : 20160411
VERSION : 3.1
// stored: AutoNumber false, SetENOAutomatically false
   VAR_INPUT
      NumSeta : UInt;
      Estado : Bool;
      MesaDeJDT02 : Bool;
   END_VAR
   VAR_OUTPUT
      Seta : "UDT_DatosSeta";
   END_VAR
   VAR_TEMP
      PunteroEventos : DWord;
      DBEventos : Word;
      NumDBEventos : UInt;
      MaxBytesDeEventos : UInt;
      NumBytes : UInt;
      ValorTMP : UDInt;
      Offset : UInt;   // Offset donde esta el Primer Dispositivo
      ValorReturn : Int;
   END_VAR
BEGIN

NETWORK
TITLE = Inicializar
////////////////////////////////////////////////////////////////////////////
// --- Inicializar Variables


////////////////////////////////////////////////////////////////////////////
// --- Control Numero de Dispositivo

      L     #NumSeta;
      L     1;
      <I;
      JC    FinalFuncion;  // Ha superado el minimo
      L     #NumSeta;
      L     "CTE_MaxDispositivosSeta";
      >I;
      JC    FinalFuncion;  // Ha superado el maximo



NETWORK
TITLE = Acciones
////////////////////////////////////////////////////////////////////////////
// --- Cambio de estado de la Seta ?

      SET;
      A     #Estado;
      AN    "DB839_DispositivosVarios".DispoSeta[#NumSeta].EstadoActual;
      JC    CambioDeEstado_Seta;

      SET;
      AN    #Estado;
      A     "DB839_DispositivosVarios".DispoSeta[#NumSeta].EstadoActual;
      JC    CambioDeEstado_Seta;


////////////////////////////////////////////////////////////////////////////
// --- Mirar si hay peticion de Estado de Seta

      SET;
      A     "DB839_DispositivosVarios".DispoSeta[#NumSeta].RefrescoDatos;
      JC    EnviarEvento_RefrescoDeDatos;  // Hay Peticion de Esatdo ?
      JU    FinalFuncion;  // No Hay Peticion de estado



////////////////////////////////////////////////////////////////////////////
// --- Ha cambiado de estado la Seta

CambioDeEstado_Seta:NOP   0;
      SET;
      A     #Estado;  // Guardar el estado de la Seta
      =     "DB839_DispositivosVarios".DispoSeta[#NumSeta].EstadoActual;

      SET;
      S     "DB839_DispositivosVarios".DispoSeta[#NumSeta].RefrescoDatos;  // Activar la Peticion de Estado de la Seta

      JU    EnviarEvento_RefrescoDeDatos;  // Mandar nuevo evento de Estado de Seta



NETWORK
TITLE = Evento de Estado de la Seta
EnviarEvento_RefrescoDeDatos:NOP   0;

////////////////////////////////////////////////////////////////////////////
// ---   Formateo del Evento de Estado del Dispositivo
// ---   * Mirar si hay sitio para generar el nuevo evento
// ---       * Inicializo NumBytes y Puntero al DB de Eventos Generados
// ---       * Calcula el tamaño de bytes que hay en el DB de Eventos Generados
// ---       * Comprobar si hay sitio para un evento más
// ---   * Formatear el evento de Estado de las Setas
////////////////////////////////////////////////////////////////////////////



////////////////////////////////////////////////////////////////////////////
// --- Inicio --> Pertenece a JDT 02 (Por defecto Pertenece a JDT01)

      L     "JDT1_NDB_EventosEmi";
      T     #DBEventos;
      T     #NumDBEventos;
      L     "JDT1_MaxBytes";
      T     #MaxBytesDeEventos;

      SET;
      AN    #MesaDeJDT02;
      JC    NoPerteneceJDT02;

      L     "JDT2_NDB_EventosEmi";
      T     #DBEventos;
      T     #NumDBEventos;
      L     "JDT2_MaxBytes";
      T     #MaxBytesDeEventos;

NoPerteneceJDT02:NOP   0;
// --- Fin --> Pertenece a JDT 02
////////////////////////////////////////////////////////////////////////////



////////////////////////////////////////////////////////////////////////////
// --- Mirar si hay sitio para generar un evento más

      L     0;
      T     #NumBytes;  // Inicializo el numero de Bytes
      T     #PunteroEventos;  // Inicializo el puntero de Eventos Generados

Inicio_BusquedaFinalEventos:NOP   0;
      OPN   DB [#DBEventos];  // Calcula el tamaño de bytes que hay en el DB
      L     DBB [#PunteroEventos];
      L     0;
      ==I;
      JC    Fin_BusquedaFinalEventos;  // Buscamos el final del DB = 0

      OPN   DB [#DBEventos];
      L     DBB [#PunteroEventos];
      L     ' ';
      ==I;
      JC    Fin_BusquedaFinalEventos;  // Buscamos el final del DB = ' '

      L     #PunteroEventos;  // Incremento de P#1.0
      L     P#1.0;
      +D;
      T     #PunteroEventos;

      JU    Inicio_BusquedaFinalEventos;  // Continuar con el siguiente posicion

Fin_BusquedaFinalEventos:NOP   0;
      L     #PunteroEventos;  // Sacamos el NumBytes Escritos
      SRD   3;
      T     #NumBytes;

      L     #NumBytes;  // Miramos si hay sitio
      L     #MaxBytesDeEventos;  // Max. que se pueden emitir, parametro
      >I;
      JC    FinalFuncion;  // No se pueden generar más eventos


////////////////////////////////////////////////////////////////////////////
// --- Formatear el evento de Estado del Dispositivo

      L     #PunteroEventos;
      LAR2;  // Puntero al DB de Eventos Generados

      TAR2;  // Mirar si es el primer evento de la lista
      L     0;
      ==I;
      JC    NoEsInicio_ListaDeEventos;  // Es el primero

      OPN   DB [#DBEventos];
      L     ',';  // Separador entre eventos ','
      T     DBB [AR2, P#0.0];
      +AR2  P#1.0;

NoEsInicio_ListaDeEventos:NOP   0;
      OPN   DB [#DBEventos];  // DB de Eventos Generados (A Emitir)
      L     '{';  // Inicio de Evento '{'
      T     DBB [AR2, P#0.0];
      +AR2  P#1.0;


////////////////////////////////////////////////////////////////////////////
      L     'STAT';  // --- Evento 'STAT'
      T     DBD [AR2, P#0.0];
      +AR2  P#4.0;


////////////////////////////////////////////////////////////////////////////
      OPN   DB [#DBEventos];
      L     '[';
      T     DBB [AR2, P#0.0];
      L     'TIPO';
      T     DBD [AR2, P#1.0];
      L     ']';
      T     DBB [AR2, P#5.0];
      +AR2  P#6.0;

      OPN   DB [#DBEventos];
      L     'SETA';  // Tipo Seta
      T     DBD [AR2, P#0.0];
      +AR2  P#4.0;


////////////////////////////////////////////////////////////////////////////
      L     '[';
      T     DBB [AR2, P#0.0];
      L     'NUME';
      T     DBD [AR2, P#1.0];
      L     ']';
      T     DBB [AR2, P#5.0];
      +AR2  P#6.0;

      L     "CTE_OffsetMesa";
      L     #NumSeta;  // Numero de la Seta
      +I;
      T     #ValorTMP;

// --- Convertir Valor a ASCII - Numero de la Baliza
      TAR2;
      SRD   3;
      T     #NumBytes;  // Miro que offset tiene la String

      CALL  "FC893_Obtener_StringDelAtributo"
      ( DB_String := #NumDBEventos,
        OffsetIni := #NumBytes,
        Valor     := #ValorTMP,
        OffsetFin := #Offset
      );  // Llamo a ObtenerStrinAtributo

      L     #Offset;
      SLD   3;
      LAR2;  // Recupero que offset tiene la String

// --- Ya esta convertido el Valor a ASCII

////////////////////////////////////////////////////////////////////////////
      OPN   DB [#DBEventos];
      L     '[';
      T     DBB [AR2, P#0.0];
      L     'ACTI';
      T     DBD [AR2, P#1.0];
      L     ']';
      T     DBB [AR2, P#5.0];
      +AR2  P#6.0;

      L     'SI';
      SET;
      A     "DB839_DispositivosVarios".DispoSeta[#NumSeta].EstadoActual;  // Activo Seta ?
      JC    EstaActiva_Seta;
      L     'NO';
EstaActiva_Seta:NOP   0;
      OPN   DB [#DBEventos];
      T     DBW [AR2, P#0.0];
      +AR2  P#2.0;


////////////////////////////////////////////////////////////////////////////
      OPN   DB [#DBEventos];
      L     '[';
      T     DBB [AR2, P#0.0];
      L     'HABI';
      T     DBD [AR2, P#1.0];
      L     ']';
      T     DBB [AR2, P#5.0];
      +AR2  P#6.0;

      L     'SI';
      SET;
      A     "DB839_DispositivosVarios".DispoSeta[#NumSeta].Habilitado;  // Habilitado ?
      JC    EstaDesHabilitada_Seta;
      L     'NO';
EstaDesHabilitada_Seta:NOP   0;
      OPN   DB [#DBEventos];
      T     DBW [AR2, P#0.0];
      +AR2  P#2.0;


////////////////////////////////////////////////////////////////////////////
      OPN   DB [#DBEventos];  // DB de Eventos Generados (A Emitir)
      L     '}';  // --- Fin de Evento '}'
      T     DBB [AR2, P#0.0];
      +AR2  P#1.0;



////////////////////////////////////////////////////////////////////////////
// --- Final del Evento

      SET;
      R     "DB839_DispositivosVarios".DispoSeta[#NumSeta].RefrescoDatos;  // Activar la Peticion de Estado de la Baliza

      JU    FinalFuncion;  //Final del Formateo del Elento



NETWORK
TITLE = Final de la Función
////////////////////////////////////////////////////////////////////////////
FinalFuncion:NOP   0;

      CALL  BLKMOV
      ( SRCBLK  := "DB839_DispositivosVarios".DispoSeta[#NumSeta],
        RET_VAL := #ValorReturn,
        DSTBLK  := #Seta
      );


END_FUNCTION

FUNCTION "FC793_GestorBarrera" : Void   // FC793, STL
{ S7_Optimized_Access := 'FALSE' }
AUTHOR : TRACKING
NAME : 20160411
VERSION : 3.1
// stored: AutoNumber false
   VAR_INPUT
      NumBarrera : UInt;
      Estado : Bool;
      MesaDeJDT02 : Bool;
   END_VAR
   VAR_OUTPUT
      Barrera : "UDT_DatosBarrera";
   END_VAR
   VAR_TEMP
      PunteroEventos : DWord;
      DBEventos : Word;
      NumDBEventos : UInt;
      MaxBytesDeEventos : UInt;
      NumBytes : UInt;
      ValorTMP : UDInt;
      Offset : UInt;   // Offset donde esta el Primer Dispositivo
      ValorReturn : Int;
   END_VAR
BEGIN

NETWORK
TITLE = Inicializar
////////////////////////////////////////////////////////////////////////////
// --- Inicializar Variables


////////////////////////////////////////////////////////////////////////////
// --- Control Numero de Dispositivo

      L     #NumBarrera;
      L     1;
      <I;
      JC    FinalFuncion;  // Ha superado el minimo
      L     #NumBarrera;
      L     "CTE_MaxDispositivosBarrera";
      >I;
      JC    FinalFuncion;  // Ha superado el maximo



NETWORK
TITLE = Acciones
////////////////////////////////////////////////////////////////////////////
// --- Cambio de estado de la Barrera ?

      SET;
      A     #Estado;
      AN    "DB839_DispositivosVarios".DispoBarrera[#NumBarrera].EstadoActual;
      JC    CambioDeEstado_Barrera;

      SET;
      AN    #Estado;
      A     "DB839_DispositivosVarios".DispoBarrera[#NumBarrera].EstadoActual;
      JC    CambioDeEstado_Barrera;


////////////////////////////////////////////////////////////////////////////
// --- Mirar si hay peticion de Estado de Barrera

      SET;
      A     "DB839_DispositivosVarios".DispoBarrera[#NumBarrera].RefrescoDatos;
      JC    EnviarEvento_RefrescoDeDatos;  // Hay Peticion de Esatdo ?
      JU    FinalFuncion;  // No Hay Peticion de estado



////////////////////////////////////////////////////////////////////////////
// --- Ha cambiado de estado la Barrera

CambioDeEstado_Barrera:NOP   0;
      SET;
      A     #Estado;  // Guardar el estado de la Barrera
      =     "DB839_DispositivosVarios".DispoBarrera[#NumBarrera].EstadoActual;

      SET;
      S     "DB839_DispositivosVarios".DispoBarrera[#NumBarrera].RefrescoDatos;  // Activar la Peticion de Estado de la Barrera

      JU    EnviarEvento_RefrescoDeDatos;  // Mandar nuevo evento de Estado de Barrera



NETWORK
TITLE = Evento de Estado de la Barrera
EnviarEvento_RefrescoDeDatos:NOP   0;

////////////////////////////////////////////////////////////////////////////
// ---   Formateo del Evento de Estado del Dispositivo
// ---   * Mirar si hay sitio para generar el nuevo evento
// ---       * Inicializo NumBytes y Puntero al DB de Eventos Generados
// ---       * Calcula el tamaño de bytes que hay en el DB de Eventos Generados
// ---       * Comprobar si hay sitio para un evento más
// ---   * Formatear el evento de Estado de las Barreras
////////////////////////////////////////////////////////////////////////////



////////////////////////////////////////////////////////////////////////////
// --- Inicio --> Pertenece a JDT 02 (Por defecto Pertenece a JDT01)

      L     "JDT1_NDB_EventosEmi";
      T     #DBEventos;
      T     #NumDBEventos;
      L     "JDT1_MaxBytes";
      T     #MaxBytesDeEventos;

      SET;
      AN    #MesaDeJDT02;
      JC    NoPerteneceJDT02;

      L     "JDT2_NDB_EventosEmi";
      T     #DBEventos;
      T     #NumDBEventos;
      L     "JDT2_MaxBytes";
      T     #MaxBytesDeEventos;

NoPerteneceJDT02:NOP   0;
// --- Fin --> Pertenece a JDT 02
////////////////////////////////////////////////////////////////////////////



////////////////////////////////////////////////////////////////////////////
// --- Mirar si hay sitio para generar un evento más

      L     0;
      T     #NumBytes;  // Inicializo el numero de Bytes
      T     #PunteroEventos;  // Inicializo el puntero de Eventos Generados

Inicio_BusquedaFinalEventos:NOP   0;
      OPN   DB [#DBEventos];  // Calcula el tamaño de bytes que hay en el DB
      L     DBB [#PunteroEventos];
      L     0;
      ==I;
      JC    Fin_BusquedaFinalEventos;  // Buscamos el final del DB = 0

      OPN   DB [#DBEventos];
      L     DBB [#PunteroEventos];
      L     ' ';
      ==I;
      JC    Fin_BusquedaFinalEventos;  // Buscamos el final del DB = ' '

      L     #PunteroEventos;  // Incremento de P#1.0
      L     P#1.0;
      +D;
      T     #PunteroEventos;

      JU    Inicio_BusquedaFinalEventos;  // Continuar con el siguiente posicion

Fin_BusquedaFinalEventos:NOP   0;
      L     #PunteroEventos;  // Sacamos el NumBytes Escritos
      SRD   3;
      T     #NumBytes;

      L     #NumBytes;  // Miramos si hay sitio
      L     #MaxBytesDeEventos;  // Max. que se pueden emitir, parametro
      >I;
      JC    FinalFuncion;  // No se pueden generar más eventos


////////////////////////////////////////////////////////////////////////////
// --- Formatear el evento de Estado del Dispositivo

      L     #PunteroEventos;
      LAR2;  // Puntero al DB de Eventos Generados

      TAR2;  // Mirar si es el primer evento de la lista
      L     0;
      ==I;
      JC    NoEsInicio_ListaDeEventos;  // Es el primero

      OPN   DB [#DBEventos];
      L     ',';  // Separador entre eventos ','
      T     DBB [AR2, P#0.0];
      +AR2  P#1.0;

NoEsInicio_ListaDeEventos:NOP   0;
      OPN   DB [#DBEventos];  // DB de Eventos Generados (A Emitir)
      L     '{';  // Inicio de Evento '{'
      T     DBB [AR2, P#0.0];
      +AR2  P#1.0;


////////////////////////////////////////////////////////////////////////////
      L     'STAT';  // --- Evento 'STAT'
      T     DBD [AR2, P#0.0];
      +AR2  P#4.0;


////////////////////////////////////////////////////////////////////////////
      OPN   DB [#DBEventos];
      L     '[';
      T     DBB [AR2, P#0.0];
      L     'TIPO';
      T     DBD [AR2, P#1.0];
      L     ']';
      T     DBB [AR2, P#5.0];
      +AR2  P#6.0;

      OPN   DB [#DBEventos];
      L     'BARR';  // Tipo Barrera
      T     DBD [AR2, P#0.0];
      +AR2  P#4.0;


////////////////////////////////////////////////////////////////////////////
      L     '[';
      T     DBB [AR2, P#0.0];
      L     'NUME';
      T     DBD [AR2, P#1.0];
      L     ']';
      T     DBB [AR2, P#5.0];
      +AR2  P#6.0;

      L     "CTE_OffsetMesa";
      L     #NumBarrera;  // Numero de la Barrera
      +I;
      T     #ValorTMP;

// --- Convertir Valor a ASCII - Numero de la Baliza
      TAR2;
      SRD   3;
      T     #NumBytes;  // Miro que offset tiene la String

      CALL  "FC893_Obtener_StringDelAtributo"
      ( DB_String := #NumDBEventos,
        OffsetIni := #NumBytes,
        Valor     := #ValorTMP,
        OffsetFin := #Offset
      );  // Llamo a ObtenerStrinAtributo

      L     #Offset;
      SLD   3;
      LAR2;  // Recupero que offset tiene la String

// --- Ya esta convertido el Valor a ASCII

////////////////////////////////////////////////////////////////////////////
      OPN   DB [#DBEventos];
      L     '[';
      T     DBB [AR2, P#0.0];
      L     'ACTI';
      T     DBD [AR2, P#1.0];
      L     ']';
      T     DBB [AR2, P#5.0];
      +AR2  P#6.0;

      L     'SI';
      SET;
      A     "DB839_DispositivosVarios".DispoBarrera[#NumBarrera].EstadoActual;  // Activo Barrera ?
      JC    EstaActiva_Barrera;
      L     'NO';
EstaActiva_Barrera:NOP   0;
      OPN   DB [#DBEventos];
      T     DBW [AR2, P#0.0];
      +AR2  P#2.0;


////////////////////////////////////////////////////////////////////////////
      OPN   DB [#DBEventos];
      L     '[';
      T     DBB [AR2, P#0.0];
      L     'HABI';
      T     DBD [AR2, P#1.0];
      L     ']';
      T     DBB [AR2, P#5.0];
      +AR2  P#6.0;

      L     'SI';
      SET;
      A     "DB839_DispositivosVarios".DispoBarrera[#NumBarrera].Habilitado;  // Habilitado ?
      JC    EstaDesHabilitada_Barrera;
      L     'NO';
EstaDesHabilitada_Barrera:NOP   0;
      OPN   DB [#DBEventos];
      T     DBW [AR2, P#0.0];
      +AR2  P#2.0;


////////////////////////////////////////////////////////////////////////////
      OPN   DB [#DBEventos];  // DB de Eventos Generados (A Emitir)
      L     '}';  // --- Fin de Evento '}'
      T     DBB [AR2, P#0.0];
      +AR2  P#1.0;



////////////////////////////////////////////////////////////////////////////
// --- Final del Evento

      SET;
      R     "DB839_DispositivosVarios".DispoBarrera[#NumBarrera].RefrescoDatos;  // Activar la Peticion de Estado de la Baliza

      JU    FinalFuncion;  //Final del Formateo del Elento



NETWORK
TITLE = Final de la Función
////////////////////////////////////////////////////////////////////////////
FinalFuncion:NOP   0;

      CALL  BLKMOV
      ( SRCBLK  := "DB839_DispositivosVarios".DispoBarrera[#NumBarrera],
        RET_VAL := #ValorReturn,
        DSTBLK  := #Barrera
      );


END_FUNCTION

FUNCTION "FC826_CalcularOrdenUT_MesaCruce" : Void   // FC826, STL
{ S7_Optimized_Access := 'FALSE' }
// stored: AutoNumber false
   VAR_INPUT
      NumeroUT : UInt;
   END_VAR
   VAR_OUTPUT
      Orden : Word;   // Orden a realizar en la MESA
      Auxiliar_01 : UInt;   // Auxiliar 01 de la Orden a realizar en la MESA
      MesaSalidaMulti : UInt;   // Auxiliar 02 de la Orden a realizar en la MESA
      Auxiliar_03 : UInt;   // Auxiliar 03 de la Orden a realizar en la MESA
      Auxiliar_04 : UInt;   // Auxiliar 04 de la Orden a realizar en la MESA
   END_VAR
   VAR_TEMP
      IndiceRutaUT : UInt;
      P_Temporal : DWord;
      MesaIntermedia : UInt;
      MesaRutaParcial : UInt;
      OrdenSalida : UInt;
      NumeroMesa : UInt;
      SiguienteUT : UInt;
      MesaEspera : UInt;
      OrdenTMP : Word;
      SinUT_EnMesa : Bool;
      RutaOK_EnMesa : Bool;
   END_VAR
BEGIN

NETWORK
TITLE = Inicializar
/////////////////////////////////////////////////////////////////////////
// Inicializaciones de las variables de los DB's

      L     0;
      T     #Orden;
      T     #OrdenTMP;
      T     #MesaSalidaMulti;
      T     #Auxiliar_01;
      T     #Auxiliar_03;
      T     #Auxiliar_04;


/////////////////////////////////////////////////////////////////////////
// Mesa Actual dentro del PLC
      L     "DB812_UTs_Control".UT[#NumeroUT].MesaActual;
      L     "CTE_OffsetMesa";
      -I;
      T     #NumeroMesa;



NETWORK
TITLE = Calcular Orden - FASE 01 >>> Ruta Para Continuar >>> Modificacion (07/05/2020)
/////////////////////////////////////////////////////////////////////////
// --- Es una Mesa de Cruce
/////////////////////////////////////////////////////////////////////////
// La mesa siguiente definida en la Mesa Actual, es una de salidas posibles
// Pero una vez encontrada la salida, debe cumplir unas condiciones:
// - Para enviar orden hay que ver si tiene que ESPERAR a que este LIBRE la
//   mesa SIGUIENTE (Mesa_Sxx) dependiendo de la salida definida
//   * Si tiene que esperar, no hacer nada
//   * Si no tiene que esperar, enviar orden y darla por tratada
//
// MODIFICACION (07/05/2020) --> Verificar si todas tienen RUTA
//
// MODIFICACION (06/05/2013) --> Nueva operativa   (ALON)
// - Buscar la mesa de salida de la ruta partiendo desde la ultima posición
//   utilizada.
//   Si no se encuentra, en esta parte de la ruta.
//   Se utilizara la ruta completa (Antigua operativa)
// OPERATIVA ANTIGUA
// - Recorrer toda la ruta, desde el principio buscando la mesa de salida
//
// - Si se envia la orden NO hay que quitar esta mesa de la ruta
//   Ya ha sido utilizada    (CAMBIO ALON - 24/10/2012)
/////////////////////////////////////////////////////////////////////////


/////////////////////////////////////////////////////////////////////////
/////////////////////////////////////////////////////////////////////////
/////////////////////////////////////////////////////////////////////////
// --- FASE 01, Mirar las rutas de las UT's de la Mesa
//     MODIFICACION AÑADIDO (07/05/2020)
      SET;
      A     "DB850_DefinicionMesas".Mesa[#NumeroMesa].ConfigMesa.RutaSalidaTodas;
      O     "DB850_DefinicionMesas".Mesa[#NumeroMesa].ConfigMesa.MultiplesCargasDeSalida;
      O     "DB850_DefinicionMesas".Mesa[#NumeroMesa].ConfigMesa.GrupoDeSalida;
      JCN   FinalControlRutaEnMesa;

// Esta parte cuidado recircular porque tiene el mismo destino
// Anulo por Ahora 2020 05 22
//      SET                        // Si tiene que recicular
//      U     #DatosUT.RecircularCarga
//      SPB   FinalControlRutaEnMesa

      CALL  "FC872_VerificarRutaEnMesa"
      ( Mesa      := #NumeroMesa,
        TestGrupo := "DB850_DefinicionMesas".Mesa[#NumeroMesa].ConfigMesa.GrupoDeSalida,
        RutaOK    := #RutaOK_EnMesa
      );

      SET;  // No tienen todas Ruta ?
      AN    #RutaOK_EnMesa;
      JC    FinalCalcularOrden;

/////////////////////////////////////////////////////////////////////////
// Tiene Ruta para Continuar - Final de FASE 02
FinalControlRutaEnMesa:NOP   0;



NETWORK
TITLE = Calcular Orden - FASE 02 >>> NUEVA OPERATIVA - Buscar por RUTA PARCIAL
/////////////////////////////////////////////////////////////////////////
/////////////////////////////////////////////////////////////////////////
/////////////////////////////////////////////////////////////////////////
// --- FASE 02, NUEVA OPERATIVA - Buscar por RUTA PARCIAL
//     MODIFICACION AÑADIDO (06/05/2013) RECIRCULACION
//     Buscar en que parte de la ruta se esta --> RUTA PARCIAL
//
//    Si no se encuentra >>> Se utilizara la Ruta Completa
//    Si se encuentra    >>> Se utilizara la Ruta Parcial


/////////////////////////////////////////////////////////////////////////
// 1. >>> Ultima Mesa tratada de la Ruta
      L     "DB812_UTs_Control".UT[#NumeroUT].MesaIntermedia;
      T     #MesaRutaParcial;


/////////////////////////////////////////////////////////////////////////
// 2. >>> Preparacion de la Ruta de la UT
      L     0;
      T     #IndiceRutaUT;


/////////////////////////////////////////////////////////////////////////
// 3. >>> Recorrer la Ruta haber si se encuentra donde se dejo
InicioBucleBusquedaInicial_EnRutaParcial:NOP   0;
      L     "DB813_UTs_Ruta".UT[#NumeroUT].Ruta[#IndiceRutaUT];
      T     #MesaIntermedia;  // Poner la nueva ruta intermedia

      L     #MesaIntermedia;  // No hay Mesa Intermedia ?
      L     0;
      ==I;  // No encontrado nada en la NUEVA OPERATIVA
      JC    FinalBucleBusqueda_EnRutaParcial;

      L     #MesaIntermedia;  // Mesa Intermedia = Mesa Ruta Parcial
      L     #MesaRutaParcial;
      ==I;  // Encontrado donde se dejo ACTIVAR NUEVA OPERATIVA
      JC    EnContradaMesa_EnRutaParcial;

      L     #MesaIntermedia;  // Se comprueba si es el Final de la Ruta
      L     "DB812_UTs_Control".UT[#NumeroUT].MesaDestino;
      ==I;  // No encontrado nada en la NUEVA OPERATIVA
      JC    FinalBucleBusqueda_EnRutaParcial;

// 3.F >>> Mesa Siguiente de la Ruta
      L     #IndiceRutaUT;
      L     1;
      +I;
      T     #IndiceRutaUT;
      JU    InicioBucleBusquedaInicial_EnRutaParcial;


/////////////////////////////////////////////////////////////////////////
// Encontrada Mesa Intermedia en RUTA PARCIAL
// NUEVA OPERATIVA (06/05/2013) RECIRCULACION
// Comprobar todas las Mesa de la Ruta PARCIAL, si esta definida alguna en la Mesa
EnContradaMesa_EnRutaParcial:NOP   0;


/////////////////////////////////////////////////////////////////////////
// 1. >>> Recorrer la Ruta haber si se encuentra, alguna Salida Definida
InicioBucleBusquedaFinal_EnRutaParcial:NOP   0;
      L     "DB813_UTs_Ruta".UT[#NumeroUT].Ruta[#IndiceRutaUT];
      T     #MesaIntermedia;  // Poner la nueva ruta intermedia

      L     #MesaIntermedia;  // No hay Mesa Intermedia ?
      L     0;
      ==I;  // No encontrado nada en la NUEVA OPERATIVA
      JC    FinalBucleBusqueda_EnRutaParcial;


/////////////////////////////////////////////////////////////////////////
// 2. >>> Comprobar cual es la mesa siguiente
//        Mesa_S01 = MesaIntermedia -> Salida por S1
//        Con Offset en la Condiguracion 28/03/2022
      L     1;  // Inicializo que sale
      T     #OrdenSalida;

      L     "DB850_DefinicionMesas".Mesa[#NumeroMesa].Mesa_S01;
//      L     "CTE_OffsetMesa"     // Mesa Correcta ?
//      +I                         // + Offset
      L     #MesaIntermedia;
      <>I;  // No es esta salida del Cruce
      JC    FinControlMesaSalida_S01_EnRutaParcial;

// --- Es esta salida del Cruce
// --- Comprobar si una Mesa de ESPERA
      SET;  // No es Salida de ESPERA ?
      AN    "DB850_DefinicionMesas".Mesa[#NumeroMesa].ConfigMesa.Espera_S01;
      JC    EnContradaMesaSalida_EnLaRuta;

// --- Mirar si Mesa_S01 esta Vacia
      L     "DB850_DefinicionMesas".Mesa[#NumeroMesa].Mesa_S01;
      L     "CTE_OffsetMesa";
      -I;  // --- Calculo de la Mesa en Espera 28/03/2022
      T     #MesaEspera;

      CALL  "FC870_MesaSinUT"
      ( Mesa  := #MesaEspera,
        SinUT := #SinUT_EnMesa
      );

      SET;  // Y la Mesa esta con UT ?
      AN    #SinUT_EnMesa;
      JC    FinalCalcularOrden;  // NO esta Vacia
      JU    EnContradaMesaSalida_EnLaRuta;

// --- Se acabo con la Mesa_S01
FinControlMesaSalida_S01_EnRutaParcial:NOP   0;


/////////////////////////////////////////////////////////////////////////
// 3. >>> Comprobar cual es la mesa siguiente
//        Mesa_S02 = MesaIntermedia -> Salida por S2
//        Con Offset en la Condiguracion 28/03/2022
      L     2;  // Inicializo que sale
      T     #OrdenSalida;

      L     "DB850_DefinicionMesas".Mesa[#NumeroMesa].Mesa_S02;
//      L     "CTE_OffsetMesa"     // Mesa Correcta ?
//      +I                         // + Offset
      L     #MesaIntermedia;
      <>I;  // No es esta salida del Cruce
      JC    FinControlMesaSalida_S02_EnRutaParcial;

// --- Es esta salida del Cruce
// --- Comprobar si una Mesa de ESPERA
      SET;  // No es Salida de ESPERA ?
      AN    "DB850_DefinicionMesas".Mesa[#NumeroMesa].ConfigMesa.Espera_S02;
      JC    EnContradaMesaSalida_EnLaRuta;

// --- Mirar si Mesa_S02 esta Vacia
      L     "DB850_DefinicionMesas".Mesa[#NumeroMesa].Mesa_S02;
      L     "CTE_OffsetMesa";
      -I;  // --- Calculo de la Mesa en Espera 28/03/2022
      T     #MesaEspera;

      CALL  "FC870_MesaSinUT"
      ( Mesa  := #MesaEspera,
        SinUT := #SinUT_EnMesa
      );

      SET;  // Y la Mesa esta con UT ?
      AN    #SinUT_EnMesa;
      JC    FinalCalcularOrden;  // NO esta Vacia
      JU    EnContradaMesaSalida_EnLaRuta;

// --- Se acabo con la Mesa_S02
FinControlMesaSalida_S02_EnRutaParcial:NOP   0;


/////////////////////////////////////////////////////////////////////////
// 4. >>> Comprobar cual es la mesa siguiente
//        Mesa_S03 = MesaIntermedia -> Salida por S3
//        Con Offset en la Condiguracion 28/03/2022
      L     3;  // Inicializo que sale por S3
      T     #OrdenSalida;

      L     "DB850_DefinicionMesas".Mesa[#NumeroMesa].Mesa_S03;
//      L     "CTE_OffsetMesa"     // Mesa Correcta ?
//      +I                         // + Offset
      L     #MesaIntermedia;
      <>I;  // No es esta salida del Cruce
      JC    FinControlMesaSalida_S03_EnRutaParcial;

// --- Es esta salida del Cruce
// --- Comprobar si una Mesa de ESPERA
      SET;  // No es Salida de ESPERA ?
      AN    "DB850_DefinicionMesas".Mesa[#NumeroMesa].ConfigMesa.Espera_S03;
      JC    EnContradaMesaSalida_EnLaRuta;

// --- Mirar si Mesa_S03 esta Vacia
      L     "DB850_DefinicionMesas".Mesa[#NumeroMesa].Mesa_S03;
      L     "CTE_OffsetMesa";
      -I;  // --- Calculo de la Mesa en Espera 28/03/2022
      T     #MesaEspera;

      CALL  "FC870_MesaSinUT"
      ( Mesa  := #MesaEspera,
        SinUT := #SinUT_EnMesa
      );

      SET;  // Y la Mesa esta con UT ?
      AN    #SinUT_EnMesa;
      JC    FinalCalcularOrden;  // NO esta Vacia
      JU    EnContradaMesaSalida_EnLaRuta;

// --- Se acabo con la Mesa_S03
FinControlMesaSalida_S03_EnRutaParcial:NOP   0;


/////////////////////////////////////////////////////////////////////////
// 5. >>> Comprobar cual es la mesa siguiente
//        Mesa_S04 = MesaIntermedia -> Salida por S4
//        Con Offset en la Condiguracion 28/03/2022
      L     4;  // Inicializo que sale
      T     #OrdenSalida;

      L     "DB850_DefinicionMesas".Mesa[#NumeroMesa].Mesa_S04;
//      L     "CTE_OffsetMesa"     // Mesa Correcta ?
//      +I                         // + Offset
      L     #MesaIntermedia;
      <>I;  // No es esta salida del Cruce
      JC    FinControlMesaSalida_S04_EnRutaParcial;

// --- Es esta salida del Cruce
// --- Comprobar si una Mesa de ESPERA
      SET;  // No es Salida de ESPERA ?
      AN    "DB850_DefinicionMesas".Mesa[#NumeroMesa].ConfigMesa.Espera_S04;
      JC    EnContradaMesaSalida_EnLaRuta;

// --- Mirar si Mesa_S04 esta Vacia
      L     "DB850_DefinicionMesas".Mesa[#NumeroMesa].Mesa_S04;
      L     "CTE_OffsetMesa";
      -I;  // --- Calculo de la Mesa en Espera 28/03/2022
      T     #MesaEspera;

      CALL  "FC870_MesaSinUT"
      ( Mesa  := #MesaEspera,
        SinUT := #SinUT_EnMesa
      );

      SET;  // Y la Mesa esta con UT ?
      AN    #SinUT_EnMesa;
      JC    FinalCalcularOrden;  // NO esta Vacia
      JU    EnContradaMesaSalida_EnLaRuta;

// --- Se acabo con la Mesa_S04
FinControlMesaSalida_S04_EnRutaParcial:NOP   0;


/////////////////////////////////////////////////////////////////////////
// 6. >>> Seguir recorriendo la RUTA PARCIAL

      L     #MesaIntermedia;  // Se comprueba si es el Final de la Ruta
      L     "DB812_UTs_Control".UT[#NumeroUT].MesaDestino;
      ==I;  // No encontrado nada en la NUEVA OPERATIVA
      JC    FinalBucleBusqueda_EnRutaParcial;

// --- Mesa Siguiente de la Ruta
      L     #IndiceRutaUT;
      L     1;
      +I;
      T     #IndiceRutaUT;
      JU    InicioBucleBusquedaFinal_EnRutaParcial;


/////////////////////////////////////////////////////////////////////////
/////////////////////////////////////////////////////////////////////////
/////////////////////////////////////////////////////////////////////////


/////////////////////////////////////////////////////////////////////////
/////////////////////////////////////////////////////////////////////////
/////////////////////////////////////////////////////////////////////////
// Final de la FASE 02 : No Encontrada >>> Utilizar RUTA COMPLETA
// RUTA PARCIAL INSUFICIENTE --> Mirar RUTA TOTAL
FinalBucleBusqueda_EnRutaParcial:NOP   0;



NETWORK
TITLE = Calcular Orden - FASE 03 >>> ANTIGUA OPERATIVA - Buscar por RUTA COMPLETA
/////////////////////////////////////////////////////////////////////////
/////////////////////////////////////////////////////////////////////////
/////////////////////////////////////////////////////////////////////////
// --- FASE 03, ANTIGUA OPERATIVA - Buscar por RUTA COMPLETA
// --- Comprobobar todas las Mesas de la Ruta,
//     si esta definida alguna en la mesa
// --- OPERATIVA (24/10/2012)


/////////////////////////////////////////////////////////////////////////
// 1. >>> Preparacion de la Ruta de la UT
      L     0;
      T     #IndiceRutaUT;


/////////////////////////////////////////////////////////////////////////
// 2. >>> Recorrer la Ruta haber si se encuentra, alguna Salida Definida
InicioBucleBusqueda_EnRutaCompleta:NOP   0;
      L     "DB813_UTs_Ruta".UT[#NumeroUT].Ruta[#IndiceRutaUT];
      T     #MesaIntermedia;  // Poner la nueva ruta intermedia

      L     #MesaIntermedia;  // No hay Mesa Intermedia ?
      L     0;
      ==I;  // No esta en Ruta, Pedir Ruta
      JC    PedirRutaNueva_FueraDeRuta;


/////////////////////////////////////////////////////////////////////////
// 3. >>> Comprobar cual es la mesa siguiente
//        Mesa_S01 = MesaIntermedia -> Salida por S1
//        Con Offset en la Condiguracion 28/03/2022
      L     1;  // Inicializo que sale
      T     #OrdenSalida;

      L     "DB850_DefinicionMesas".Mesa[#NumeroMesa].Mesa_S01;
//      L     "CTE_OffsetMesa"     // Mesa Correcta ?
//      +I                         // + Offset
      L     #MesaIntermedia;
      <>I;  // No es esta salida del Cruce
      JC    FinControlMesaSalida_S01_EnRutaCompleta;

// --- Es esta salida del Cruce
// --- Comprobar si una Mesa de ESPERA
      SET;  // No es Salida de ESPERA ?
      AN    "DB850_DefinicionMesas".Mesa[#NumeroMesa].ConfigMesa.Espera_S01;
      JC    EnContradaMesaSalida_EnLaRuta;

// --- Mirar si Mesa_S01 esta Vacia
      L     "DB850_DefinicionMesas".Mesa[#NumeroMesa].Mesa_S01;
      L     "CTE_OffsetMesa";
      -I;  // --- Calculo de la Mesa en Espera 28/03/2022
      T     #MesaEspera;

      CALL  "FC870_MesaSinUT"
      ( Mesa  := #MesaEspera,
        SinUT := #SinUT_EnMesa
      );

      SET;  // Y la Mesa esta con UT ?
      AN    #SinUT_EnMesa;
      JC    FinalCalcularOrden;  // NO esta Vacia
      JU    EnContradaMesaSalida_EnLaRuta;

// --- Se acabo con la Mesa_S01
FinControlMesaSalida_S01_EnRutaCompleta:NOP   0;


/////////////////////////////////////////////////////////////////////////
// 4. >>> Comprobar cual es la mesa siguiente
//        Mesa_S02 = MesaIntermedia -> Salida por S2
//        Con Offset en la Condiguracion 28/03/2022
      L     2;  // Inicializo que sale
      T     #OrdenSalida;

      L     "DB850_DefinicionMesas".Mesa[#NumeroMesa].Mesa_S02;
//      L     "CTE_OffsetMesa"     // Mesa Correcta ?
//      +I                         // + Offset
      L     #MesaIntermedia;
      <>I;  // No es esta salida del Cruce
      JC    FinControlMesaSalida_S02_EnRutaCompleta;

// --- Es esta salida del Cruce
// --- Comprobar si una Mesa de ESPERA
      SET;  // No es Salida de ESPERA ?
      AN    "DB850_DefinicionMesas".Mesa[#NumeroMesa].ConfigMesa.Espera_S02;
      JC    EnContradaMesaSalida_EnLaRuta;

// --- Mirar si Mesa_S02 esta Vacia
      L     "DB850_DefinicionMesas".Mesa[#NumeroMesa].Mesa_S02;
      L     "CTE_OffsetMesa";
      -I;  // --- Calculo de la Mesa en Espera 28/03/2022
      T     #MesaEspera;

      CALL  "FC870_MesaSinUT"
      ( Mesa  := #MesaEspera,
        SinUT := #SinUT_EnMesa
      );

      SET;  // Y la Mesa esta con UT ?
      AN    #SinUT_EnMesa;
      JC    FinalCalcularOrden;  // NO esta Vacia
      JU    EnContradaMesaSalida_EnLaRuta;

// --- Se acabo con la Mesa_S02
FinControlMesaSalida_S02_EnRutaCompleta:NOP   0;


/////////////////////////////////////////////////////////////////////////
// 5. >>> Comprobar cual es la mesa siguiente
//        Mesa_S03 = MesaIntermedia -> Salida por S3
//        Con Offset en la Condiguracion 28/03/2022
      L     3;  // Inicializo que sale por S3
      T     #OrdenSalida;

      L     "DB850_DefinicionMesas".Mesa[#NumeroMesa].Mesa_S03;
//      L     "CTE_OffsetMesa"     // Mesa Correcta ?
//      +I                         // + Offset
      L     #MesaIntermedia;
      <>I;  // No es esta salida del Cruce
      JC    FinControlMesaSalida_S03_EnRutaCompleta;

// --- Es esta salida del Cruce
// --- Comprobar si una Mesa de ESPERA
      SET;  // No es Salida de ESPERA ?
      AN    "DB850_DefinicionMesas".Mesa[#NumeroMesa].ConfigMesa.Espera_S03;
      JC    EnContradaMesaSalida_EnLaRuta;

// --- Mirar si Mesa_S03 esta Vacia
      L     "DB850_DefinicionMesas".Mesa[#NumeroMesa].Mesa_S03;
      L     "CTE_OffsetMesa";
      -I;  // --- Calculo de la Mesa en Espera 28/03/2022
      T     #MesaEspera;

      CALL  "FC870_MesaSinUT"
      ( Mesa  := #MesaEspera,
        SinUT := #SinUT_EnMesa
      );

      SET;  // Y la Mesa esta con UT ?
      AN    #SinUT_EnMesa;
      JC    FinalCalcularOrden;  // NO esta Vacia
      JU    EnContradaMesaSalida_EnLaRuta;

// --- Se acabo con la Mesa_S03
FinControlMesaSalida_S03_EnRutaCompleta:NOP   0;


/////////////////////////////////////////////////////////////////////////
// 6. >>> Comprobar cual es la mesa siguiente
//        Mesa_S04 = MesaIntermedia -> Salida por S4
//        Con Offset en la Condiguracion 28/03/2022
      L     4;  // Inicializo que sale
      T     #OrdenSalida;

      L     "DB850_DefinicionMesas".Mesa[#NumeroMesa].Mesa_S04;
//      L     "CTE_OffsetMesa"     // Mesa Correcta ?
//      +I                         // + Offset
      L     #MesaIntermedia;
      <>I;  // No es esta salida del Cruce
      JC    FinControlMesaSalida_S04_EnRutaCompleta;

// --- Es esta salida del Cruce
// --- Comprobar si una Mesa de ESPERA
      SET;  // No es Salida de ESPERA ?
      AN    "DB850_DefinicionMesas".Mesa[#NumeroMesa].ConfigMesa.Espera_S04;
      JC    EnContradaMesaSalida_EnLaRuta;

// --- Mirar si Mesa_S04 esta Vacia
      L     "DB850_DefinicionMesas".Mesa[#NumeroMesa].Mesa_S04;
      L     "CTE_OffsetMesa";
      -I;  // --- Calculo de la Mesa en Espera 28/03/2022
      T     #MesaEspera;

      CALL  "FC870_MesaSinUT"
      ( Mesa  := #MesaEspera,
        SinUT := #SinUT_EnMesa
      );

      SET;  // Y la Mesa esta con UT ?
      AN    #SinUT_EnMesa;
      JC    FinalCalcularOrden;  // NO esta Vacia
      JU    EnContradaMesaSalida_EnLaRuta;

// --- Se acabo con la Mesa_S04
FinControlMesaSalida_S04_EnRutaCompleta:NOP   0;


/////////////////////////////////////////////////////////////////////////
// 7. >>> Seguir recorriendo la RUTA Completa

      L     #MesaIntermedia;  // Se comprueba si es el Final de la Ruta
      L     "DB812_UTs_Control".UT[#NumeroUT].MesaDestino;
      ==I;  // No encontrado nada en la NUEVA OPERATIVA
      JC    PedirRutaNueva_FueraDeRuta;

// --- Mesa Siguiente de la Ruta
      L     #IndiceRutaUT;
      L     1;
      +I;
      T     #IndiceRutaUT;
      JU    InicioBucleBusqueda_EnRutaCompleta;


/////////////////////////////////////////////////////////////////////////
/////////////////////////////////////////////////////////////////////////
/////////////////////////////////////////////////////////////////////////


/////////////////////////////////////////////////////////////////////////
/////////////////////////////////////////////////////////////////////////
/////////////////////////////////////////////////////////////////////////
// Final de la FASE 03 : Encontrada Mesa de Salida
FinalBucleBusqueda_EnRutaCompleta:NOP   0;
      JU    EnContradaMesaSalida_EnLaRuta;



NETWORK
TITLE = Calcular Orden - FASE 04 >>> Encontrada Mesa de Salida En la Ruta
/////////////////////////////////////////////////////////////////////////
/////////////////////////////////////////////////////////////////////////
/////////////////////////////////////////////////////////////////////////
// --- FASE 04, Encontrada Mesa de Salida En la Ruta
// --- Primero, doy por tratada la causa
// --- Segundo, Activarse la Mesa de Salida que Corresponda "OrdenSalida"
EnContradaMesaSalida_EnLaRuta:NOP   0;


/////////////////////////////////////////////////////////////////////////
// 1 >>> Doy por tratada la Mesa la Primera de la Mesa
      L     0;  // Dar por tratada
      T     "DB812_UTs_Control".UT[#NumeroUT].EstadoRecepcionUT;
      T     "DB812_UTs_Control".UT[#NumeroUT].EstadoEventoRecibido;

      L     #MesaIntermedia;
      T     "DB812_UTs_Control".UT[#NumeroUT].MesaIntermedia;

      SET;  // Reset - Recircular la Carga - Memoria del Retirar
      R     "DB812_UTs_Control".UT[#NumeroUT].AtributosDeLaUT.RecircularCarga;


/////////////////////////////////////////////////////////////////////////
// 2 >>> Si hay que darla por tratadas todas las de la Mesa

      SET;  // Hay que Recorrer el Resto de UTs de la Mesa
      AN    "DB850_DefinicionMesas".Mesa[#NumeroMesa].ConfigMesa.MultiplesCargasDeSalida;
      AN    "DB850_DefinicionMesas".Mesa[#NumeroMesa].ConfigMesa.GrupoDeSalida;
      JC    FinalBucleUTs_EnMesa;

      L     "DB812_UTs_Control".UT[#NumeroUT].UT_SiguienteMesa;
      T     #SiguienteUT;


InicioBucleUTs_EnMesa:NOP   0;
      L     #SiguienteUT;
      L     0;
      ==I;  // Hay mas UT's
      JC    FinalBucleUTs_EnMesa;

// Testear Grupo ?
      SET;
      AN    "DB850_DefinicionMesas".Mesa[#NumeroMesa].ConfigMesa.GrupoDeSalida;
      JC    ContinuarBucleUTs_EnMesa;

// Dar por tratado solo lo del mismo Grupo
// Grupo Primera UT == Grupo de la Siguiente
      L     "DB812_UTs_Control".UT[#NumeroUT].Grupo;
      L     "DB812_UTs_Control".UT[#SiguienteUT].Grupo;
      <>I;
      JC    FinalBucleUTs_EnMesa;

// Dar por tratada la Siguinete UT
ContinuarBucleUTs_EnMesa:NOP   0;
      L     0;  // Dar por tratada
      T     "DB812_UTs_Control".UT[#SiguienteUT].EstadoRecepcionUT;
      T     "DB812_UTs_Control".UT[#SiguienteUT].EstadoEventoRecibido;

      L     #MesaIntermedia;
      T     "DB812_UTs_Control".UT[#SiguienteUT].MesaIntermedia;

      SET;  // Reset - Recircular la Carga - Memoria del Retirar
      R     "DB812_UTs_Control".UT[#NumeroUT].AtributosDeLaUT.RecircularCarga;

      L     "DB812_UTs_Control".UT[#SiguienteUT].UT_SiguienteMesa;
      T     #SiguienteUT;
      JU    InicioBucleUTs_EnMesa;


/////////////////////////////////////////////////////////////////////////
// 2. >>> Final del Bucle
FinalBucleUTs_EnMesa:NOP   0;


/////////////////////////////////////////////////////////////////////////
// 3. >>>   Activarse la Mesa de Salida que Corresponda
//          En variable "OrdenSalida"

      L     #OrdenSalida;
      JL    SinOrden_Defecto;

// 3.1. Distribucion de la Orden de Salida
      JU    SinOrden_Defecto;  // OrdenSalida = 0
      JU    OrdenSalida_S01;  // OrdenSalida = 1
      JU    OrdenSalida_S02;  // OrdenSalida = 2
      JU    OrdenSalida_S03;  // OrdenSalida = 3
      JU    OrdenSalida_S04;  // OrdenSalida = 4

// 3.2. >>>> CUIDADO si llega aqui MALO es IMPOSIBLE
SinOrden_Defecto:NOP   0;
      JU    FinalCalcularOrden;



NETWORK
TITLE = Control - No existe Mesa de Salida - FUERA de RUTA
/////////////////////////////////////////////////////////////////////////
// --- No existe Mesa de Salida posible
//     La UT esta FUERA de RUTA
//     Realiazar, Evento de Pedir Ruta

PedirRutaNueva_FueraDeRuta:NOP   0;
      L     "DB812_UTs_Control".UT[#NumeroUT].EstadoGeneralUT;
      L     0;
      <>I;  //NO esta LIBRE?
      JC    FinalCalcularOrden;

      L     26;  // 26 - Generar Evento Pedir Ruta (FUERA DE RUTA)
      T     "DB812_UTs_Control".UT[#NumeroUT].EstadoGeneralUT;
      L     0;  // Dar por tratada
      T     "DB812_UTs_Control".UT[#NumeroUT].EstadoRecepcionUT;

      JU    FinalCalcularOrden;



NETWORK
TITLE = Generar Orden de Salida
/////////////////////////////////////////////////////////////////////////
/////////////////////////////////////////////////////////////////////////
// --- Ordenes a enviar dependiendo por donde sale
// --- Salida por S01
OrdenSalida_S01:NOP   0;
      L     P##OrdenTMP;
      L     P#0.1;
      +D;
      T     #P_Temporal;

      SET;  // Orden -> Activar Bit 1
      S     L [#P_Temporal];
      JU    FinalOrdenSalida;


/////////////////////////////////////////////////////////////////////////
/////////////////////////////////////////////////////////////////////////
// --- Ordenes a enviar dependiendo por donde sale
// --- Salida por S02
OrdenSalida_S02:NOP   0;
      L     P##OrdenTMP;
      L     P#0.2;
      +D;
      T     #P_Temporal;

      SET;  // Orden -> Activar Bit 2
      S     L [#P_Temporal];
      JU    FinalOrdenSalida;


/////////////////////////////////////////////////////////////////////////
/////////////////////////////////////////////////////////////////////////
// --- Ordenes a enviar dependiendo por donde sale
// --- Salida por S03
OrdenSalida_S03:NOP   0;
      L     P##OrdenTMP;
      L     P#0.3;
      +D;
      T     #P_Temporal;

      SET;  // Orden -> Activar Bit 3
      S     L [#P_Temporal];
      JU    FinalOrdenSalida;


/////////////////////////////////////////////////////////////////////////
/////////////////////////////////////////////////////////////////////////
// --- Ordenes a enviar dependiendo por donde sale
// --- Salida por S04
OrdenSalida_S04:NOP   0;
      L     P##OrdenTMP;
      L     P#0.4;
      +D;
      T     #P_Temporal;

      SET;  // Orden -> Activar Bit 4
      S     L [#P_Temporal];
      JU    FinalOrdenSalida;



/////////////////////////////////////////////////////////////////////////
/////////////////////////////////////////////////////////////////////////
// --- Ordenes a enviar dependiendo por donde sale
// --- Salida por Defecto
OrdenSalida_Defecto:NOP   0;
      L     P##OrdenTMP;
      L     P#0.5;
      +D;
      T     #P_Temporal;

      SET;  // Orden -> Activar Bit 5
      S     L [#P_Temporal];
      JU    FinalOrdenSalida;


/////////////////////////////////////////////////////////////////////////
/////////////////////////////////////////////////////////////////////////
// No Existen mas posibilidades
FinalOrdenSalida:NOP   0;



NETWORK
TITLE = Final de Calcular Orden
/////////a////////////////////////////////////////////////////////////////
// Finalizar la Funcion
FinalCalcularOrden:NOP   0;

      L     #OrdenTMP;
      T     #Orden;


END_FUNCTION

FUNCTION "FC834_GestorMaquinaSimple" : Void   // FC834, LAD
TITLE = Tracking de la Maquina Base
{ S7_Optimized_Access := 'FALSE' }
AUTHOR : TRACKING
NAME : 20160525
VERSION : 3.1
// - Inicializar
// - Recoger datos necesarios del Sistema
// 
// - Dispositivo Maquina
//   + Gestion de Estado
//   + Gestion de Control de Reset
//   + Gestion de Control de Paro Blando
//   + Gestion de Control de Errores
// 
// - Operaciones propias de la Maquina
// 
// - Cierre de protocolo de la Maquina
// - Actualizar datos del Sistema
// stored: AutoNumber false, SetENOAutomatically false
   VAR_INPUT
      DB_VIMaquina : DB_ANY;   // DB de la Maquina
      EstadoZonaMesa : "EstadoZona";   // Estado de la Zona Mesa Asociada a la Mesa
      NumMaquina : UInt;   // Numero de la Maquina
      RearmeError : Bool;   // Rearme de Errores Adicionales
      ManualReset : Bool;   // Resetear la Maquina desde el exterior
      FinReset : Bool;   // Reset Finalizado del VI Maquina
      ManualParoBlando : Bool;   // Paro Blando de la Mauina desde el exterior
      FinParoBlando : Bool;   // Paro Blando Finalizado del VI Maquina
   END_VAR
   VAR_TEMP
      PunteroDBVIMaquina : Any;
      P_EstadoVI : DWord;
      PunteroDBTMP : DWord;
      DBEstadoVI : Word;
      CodigoErrorMesa : UDInt;   // Error (Código) de la Mesa (Dispositivo)
      NumeroErrorVI : UInt;
      Maquina : UInt;   // Numero de Maquina dentro del PLC
      ByteTMP : Byte;
      ReturnValor : Int;
      TMPFinReset_NOK : Bool;
      TMPFinParoBlando_NOK : Bool;
      FlancoAuto : Bool;
      FlancoManual : Bool;
      FlancoMarcha : Bool;
      FlancoParo : Bool;
      FlancoReset : Bool;
      FlancoParoBlando : Bool;
      FinResetTMP : Bool;
      FinParoBlandoTMP : Bool;
   END_VAR
BEGIN

NETWORK
TITLE = Inicializar
/////////////////////////////////////////////////////////////////////////////
// --- Inicializar las Variables

      L     #NumMaquina;
      T     #Maquina;


/////////////////////////////////////////////////////////////////////////////
// --- Estado Mesa - Salida Inicializar a cero - Zona

      L     0;  // Que rellenar en el DB
      T     #ByteTMP;

      CALL  FILL
      ( BVAL    := #ByteTMP,
        RET_VAL := #ReturnValor,
        BLK     := "DB903_Estado_ZonaMaquina".EstadoMaquina[#Maquina]
      );  // Reseteo el la zona temp



NETWORK
TITLE = Gestion del Estado de la Maquina - Inicial
/////////////////////////////////////////////////////////////////////////////
// --- Flancos de los estados de la Maquina

      SET;
      A     #EstadoZonaMesa.Automatico_CBx;
      FP    "DB832_Maquinas".Maquinas[#Maquina].Memorias.MFL_Auto;  // Memo Automatico
      =     #FlancoAuto;

      SET;
      A     #EstadoZonaMesa.Manual_CBx;
      FP    "DB832_Maquinas".Maquinas[#Maquina].Memorias.MFL_Manual;  // Memo Manual
      =     #FlancoManual;

      SET;
      A     #EstadoZonaMesa.Marcha_CBx;
      FP    "DB832_Maquinas".Maquinas[#Maquina].Memorias.MFL_Marcha;  // Memo Marcha
      =     #FlancoMarcha;

      SET;
      A     #EstadoZonaMesa.Paro_CBx;
      FP    "DB832_Maquinas".Maquinas[#Maquina].Memorias.MFL_Paro;  // Memo Paro
      =     #FlancoParo;



NETWORK
TITLE = ---- Automatico, Manual
/////////////////////////////////////////////////////////////////////////////
// --- Estado de la Maquina
// --- Nota: Si cambia Auto/Remoto/Manual se pasa a Paro
// --- Nota: Si hay Marcha solo si esta en Automatico o Remoto
// ---       nunca en Manual

/////////////////////////////////////////////////////////////////////////////
// --- Maquina en Automatico (Estado: Automatico y Paro)
// --- Condicion: si la Zona Mesa esta en Automatico
      SET;
      A(;
      O     #FlancoAuto;  // Automatico de la Zona Mesa
      O     "DB841_Recepcion".DispoMaquina[#Maquina].Protocolo.Automatico;  // Automatico de la Orden Maquina
      );
      A     #EstadoZonaMesa.Automatico_CBx;  // Condicion
      JCN   NoEsta_EstadoDeLlaveEnAutomatico;

      SET;
      S     "DB840_Emision".DispoMaquina[#Maquina].Protocolo.Automatico;  // Poner en Automatico
      R     "DB840_Emision".DispoMaquina[#Maquina].Protocolo.Manual;

      JU    Final_EstadoDeLLave;

NoEsta_EstadoDeLlaveEnAutomatico:NOP   0;


/////////////////////////////////////////////////////////////////////////////
// --- Maquina en Manual (Estado: Manual y Paro)
// --- Condicion: Ninguna

      SET;
      A(;
      O     #FlancoManual;  // Manual de la Zona Mesa
      O     "DB841_Recepcion".DispoMaquina[#Maquina].Protocolo.Manual;  // Manual de la Orden Maquina
      );
      JCN   NoEsta_EstadoDeLlaveEnManual;

      SET;
      R     "DB840_Emision".DispoMaquina[#Maquina].Protocolo.Automatico;  // Poner en Manual
      S     "DB840_Emision".DispoMaquina[#Maquina].Protocolo.Manual;

      JU    Final_EstadoDeLLave;

NoEsta_EstadoDeLlaveEnManual:NOP   0;


/////////////////////////////////////////////////////////////////////////////
// --- Final Control de Llave de Mesa (En Automatico y En Manual)
Final_EstadoDeLLave:NOP   0;



NETWORK
TITLE = ---- Marcha, Paro
/////////////////////////////////////////////////////////////////////////////
// --- Maquina en Marcha
// --- Condicion: si esta la Maquina en Automatico o Remoto
// ---            si esta la Zona Mesa en Marcha

      SET;
      A(;
      O     #FlancoMarcha;  // Marcha de la Zona Mesa
      O     "DB841_Recepcion".DispoMaquina[#Maquina].Protocolo.Marcha;  // Marcha de la Orden Maquina
      );
      AN    #EstadoZonaMesa.Manual_CBx;  // Condiciones
      A     #EstadoZonaMesa.Marcha_CBx;

      AN    "DB840_Emision".DispoMaquina[#Maquina].Protocolo.Reset_Realizandose;
      JCN   NoEsta_EstadoDeMesaEnMarcha;

      SET;
      S     "DB840_Emision".DispoMaquina[#Maquina].Protocolo.Marcha;  // Poner en Marcha
      R     "DB840_Emision".DispoMaquina[#Maquina].Protocolo.Paro;
      R     "DB840_Emision".DispoMaquina[#Maquina].Protocolo.ParoBlando_Realizandose;  // Resetear Variables
      R     "DB840_Emision".DispoMaquina[#Maquina].Protocolo.ParoBlandoNOK;  // De Paro Blando
      R     "DB840_Emision".DispoMaquina[#Maquina].Protocolo.ParoBlandoOK;

      JU    Final_EstadoDeMesa;

NoEsta_EstadoDeMesaEnMarcha:NOP   0;


/////////////////////////////////////////////////////////////////////////////
// --- Maquina en Paro
// --- Condicion: Ninguna

      SET;
      A     #FlancoParo;  // Paro de la Zona Mesa
      O     "DB841_Recepcion".DispoMaquina[#Maquina].Protocolo.Paro;  // Paro de la Orden Maquina

      O     #FlancoAuto;  // Automatcio de la Zona Mesa
      O     #FlancoManual;  // Manual de la Zona Mesa

      O     "DB841_Recepcion".DispoMaquina[#Maquina].Protocolo.Automatico;  // Automatico de la Orden Maquina
      O     "DB841_Recepcion".DispoMaquina[#Maquina].Protocolo.Manual;  // Manual de la Orden Maquina

      JCN   NoEsta_EstadoDeMesaEnParo;

      SET;
      R     "DB840_Emision".DispoMaquina[#Maquina].Protocolo.Marcha;  // Poner en Paro
      S     "DB840_Emision".DispoMaquina[#Maquina].Protocolo.Paro;

NoEsta_EstadoDeMesaEnParo:NOP   0;


/////////////////////////////////////////////////////////////////////////////
// --- Final del control de Estado de Mesa (Marcha, Paro)
Final_EstadoDeMesa:NOP   0;




NETWORK
TITLE = Temporizador de Reset y Paro Blando NOK
/////////////////////////////////////////////////////////////////////////////
// --- Temporizador de Fin de Reset NOK

      CALL  "FC899_TMP"
      ( Temporizar     := "DB840_Emision".DispoMaquina[#Maquina].Protocolo.Reset_Realizandose,
        Valor_Tiempo   := "CTE_TMPEsperaFinReset",
        Base_tiempo_ms := 1000,
        Tiempo_OK      := #TMPFinReset_NOK,
        Valor_Actual   := "DB832_Maquinas".Maquinas[#Maquina].TMP_Reset
      );


/////////////////////////////////////////////////////////////////////////////
// --- Temporizador de Fin de ParoBlando NOK

      CALL  "FC899_TMP"
      ( Temporizar     := "DB840_Emision".DispoMaquina[#Maquina].Protocolo.ParoBlando_Realizandose,
        Valor_Tiempo   := "CTE_TMPEsperaFinReset",
        Base_tiempo_ms := 1000,
        Tiempo_OK      := #TMPFinParoBlando_NOK,
        Valor_Actual   := "DB832_Maquinas".Maquinas[#Maquina].TMP_ParoBlando
      );



NETWORK
TITLE = Gestion de Control de Reset
/////////////////////////////////////////////////////////////////////////////
// --- Flanco de Activacion de Reset

      SET;
      A     #EstadoZonaMesa.Resetear_CBx;  // Por la Zona Mesa
      O     #ManualReset;  // Manualmente (Exterior)
      O     "DB841_Recepcion".DispoMaquina[#Maquina].Protocolo.Reset;  // Por la Orden
      FP    "DB832_Maquinas".Maquinas[#Maquina].Memorias.MFL_Reset;  // Memo Reset
      =     #FlancoReset;

      SET;
      A     #FinReset;  // No hace caso si no hay Reset
      A     "DB904_Estado_Maquinas".EstadoVI[#Maquina].Fin_VI;
      A     "DB840_Emision".DispoMaquina[#Maquina].Protocolo.Reset_Realizandose;
      =     #FinResetTMP;

/////////////////////////////////////////////////////////////////////////////
// --- Activacion del Proceso de Reset

      SET;
      AN    #FlancoReset;
      JC    SistemaReset_Gestion;  // Hay que Realizar el Reset ?

      SET;
      A     "DB840_Emision".DispoMaquina[#Maquina].Protocolo.Marcha;
      JC    ResetImposible;


/////////////////////////////////////////////////////////////////////////////
// --- Se ha producido un Reset valido (Reseteo de las variables)

      SET;
      S     "DB840_Emision".DispoMaquina[#Maquina].Protocolo.Reset_Realizandose;  // Reseteando la Maquina
      R     "DB840_Emision".DispoMaquina[#Maquina].Protocolo.ParoBlando_Realizandose;  // Resetear Variables
      R     "DB840_Emision".DispoMaquina[#Maquina].Protocolo.ParoBlandoNOK;  // De Paro Blando
      R     "DB840_Emision".DispoMaquina[#Maquina].Protocolo.ParoBlandoOK;

      L     0;  // Reseteo el Status de Trabajo
      T     "DB832_Maquinas".Maquinas[#Maquina].MemoriaEstado;  // NuevoStatusTrabajo


/////////////////////////////////////////////////////////////////////////////
// --- Reseteo - DB del Vehiculo Inteligente

      OPN   #DB_VIMaquina;  // Abro el DB a resetear
      LAR1  P##PunteroDBVIMaquina;  // Preparar Puntero Any
      L     B#16#10;  // ID de Sintasis
      T     LB [AR1, P#0.0];
      L     B#16#2;  // Tipo de Datos
      T     LB [AR1, P#1.0];
      L     DBLG;  // Longitud del DB
      T     LW [AR1, P#2.0];
      L     DBNO;  // Numero de DB
      T     LW [AR1, P#4.0];
      L     0;
      SLW   3;
      T     LD [AR1, P#6.0];
      L     B#16#84;  // Indico el tipo DB
      T     LB [AR1, P#6.0];

      L     0;  // Que rellenar en el DB
      T     #ByteTMP;
      CALL  FILL
      ( BVAL    := #ByteTMP,
        RET_VAL := #ReturnValor,
        BLK     := #PunteroDBVIMaquina
      );  // Reseteo el DB


/////////////////////////////////////////////////////////////////////////////
// --- Reseteo - Estado del Vehiculo Inteligente

      L     0;  // Reseteo del Estado del VI
      T     #ByteTMP;
      CALL  FILL
      ( BVAL    := #ByteTMP,
        RET_VAL := #ReturnValor,
        BLK     := "DB904_Estado_Maquinas".EstadoVI[#Maquina]
      );


/////////////////////////////////////////////////////////////////////////////
// --- No hay más que resetar
      JU    SistemaReset_Gestion;


/////////////////////////////////////////////////////////////////////////////
// --- Reset Imposible

ResetImposible:NOP   0;
      SET;
      S     "DB840_Emision".DispoMaquina[#Maquina].Protocolo.ResetNOK;  // Activa del Bit Reset Imposible
      R     "DB840_Emision".DispoMaquina[#Maquina].Protocolo.ResetOK;  // Desactiva el Bit de Reset OK
      R     "DB840_Emision".DispoMaquina[#Maquina].Protocolo.Reset_Realizandose;

      JU    SistemaReset_Gestion;


/////////////////////////////////////////////////////////////////////////////
/////////////////////////////////////////////////////////////////////////////
/////////////////////////////////////////////////////////////////////////////
/////////////////////////////////////////////////////////////////////////////
// --- Gestion de Reset
SistemaReset_Gestion:NOP   0;
      SET;
      AN    "DB840_Emision".DispoMaquina[#Maquina].Protocolo.Reset_Realizandose;
      JC    SistemaReset_Fin;

      SET;
      AN    #EstadoZonaMesa.Resetear_CBx;  // Por la Zona
      AN    #EstadoZonaMesa.PerReset_CBx;
      AN    #ManualReset;  // Manualmente (Exterior)
      AN    "DB841_Recepcion".DispoMaquina[#Maquina].Protocolo.Reset;  // Por la Orden
      A     "DB841_Recepcion".DispoMaquina[#Maquina].Protocolo.EmiOK;  // Avisado el JdT ?
      JCN   SistemaReset_Continuar;


